gfCNCPoint5[3628] = {X 478.2330, Y 32.3647, Z -6.3333, A 0.000, B 0.000, C 0.000 }
gfCNCPoint5[3629] = {X 476.9689, Y 31.4976, Z -6.3333, A 0.000, B 0.000, C 0.000 }
gfCNCPoint5[3630] = {X 475.8319, Y 30.4695, Z -6.3333, A 0.000, B 0.000, C 0.000 }
gfCNCPoint5[3631] = {X 474.8423, Y 29.2987, Z -6.3333, A 0.000, B 0.000, C 0.000 }
gfCNCPoint5[3632] = {X 474.0180, Y 28.0063, Z -6.3333, A 0.000, B 0.000, C 0.000 }
gfCNCPoint5[3633] = {X 473.3736, Y 26.6154, Z -6.3333, A 0.000, B 0.000, C 0.000 }
gfCNCPoint5[3634] = {X 472.9207, Y 25.1509, Z -6.3333, A 0.000, B 0.000, C 0.000 }
gfCNCPoint5[3635] = {X 472.6068, Y 23.4678, Z -6.3333, A 0.000, B 0.000, C 0.000 }
gfCNCPoint5[3636] = {X 472.4665, Y 21.7615, Z -6.3333, A 0.000, B 0.000, C 0.000 }
gfCNCPoint5[3637] = {X 472.5012, Y 20.0497, Z -6.3333, A 0.000, B 0.000, C 0.000 }
gfCNCPoint5[3638] = {X 472.7106, Y 18.3505, Z -6.3333, A 0.000, B 0.000, C 0.000 }
gfCNCPoint5[3639] = {X 473.0925, Y 16.6815, Z -6.3333, A 0.000, B 0.000, C 0.000 }
gfCNCPoint5[3640] = {X 473.6354, Y 15.1666, Z -6.3333, A 0.000, B 0.000, C 0.000 }
gfCNCPoint5[3641] = {X 474.3788, Y 13.7394, Z -6.3333, A 0.000, B 0.000, C 0.000 }
gfCNCPoint5[3642] = {X 475.3090, Y 12.4262, Z -6.3333, A 0.000, B 0.000, C 0.000 }
gfCNCPoint5[3643] = {X 476.4087, Y 11.2513, Z -6.3333, A 0.000, B 0.000, C 0.000 }
gfCNCPoint5[3644] = {X 477.6577, Y 10.2366, Z -6.3333, A 0.000, B 0.000, C 0.000 }
gfCNCPoint5[3645] = {X 479.0328, Y 9.4006, Z -6.3333, A 0.000, B 0.000, C 0.000 }
gfCNCPoint5[3646] = {X 480.5086, Y 8.7590, Z -6.3333, A 0.000, B 0.000, C 0.000 }
gfCNCPoint5[3647] = {X 482.0578, Y 8.3236, Z -6.3333, A 0.000, B 0.000, C 0.000 }
gfCNCPoint5[3648] = {X 484.1552, Y 7.9970, Z -6.3333, A 0.000, B 0.000, C 0.000 }
gfCNCPoint5[3649] = {X 486.2746, Y 7.8821, Z -6.3333, A 0.000, B 0.000, C 0.000 }
gfCNCPoint5[3650] = {X 486.9679, Y 7.8699, Z -6.3333, A 0.000, B 0.000, C 0.000 }
gfCNCPoint5[3651] = {X 492.3835, Y 7.8699, Z -6.3333, A 0.000, B 0.000, C 0.000 }
gfCNCPoint5[3652] = {X 492.3835, Y 3.8699, Z -6.3333, A 0.000, B 0.000, C 0.000 }
gfCNCPoint5[3653] = {X 492.3835, Y 7.9499, Z -6.3333, A 0.000, B 0.000, C 0.000 }
gfCNCPoint5[3654] = {X 502.2063, Y 7.9499, Z -6.3333, A 0.000, B 0.000, C 0.000 }
gfCNCPoint5[3655] = {X 502.7389, Y 7.9541, Z -6.3333, A 0.000, B 0.000, C 0.000 }
gfCNCPoint5[3656] = {X 503.6731, Y 8.0662, Z -6.3333, A 0.000, B 0.000, C 0.000 }
gfCNCPoint5[3657] = {X 504.5592, Y 8.3824, Z -6.3333, A 0.000, B 0.000, C 0.000 }
gfCNCPoint5[3658] = {X 505.3534, Y 8.8870, Z -6.3333, A 0.000, B 0.000, C 0.000 }
gfCNCPoint5[3659] = {X 506.0160, Y 9.5548, Z -6.3333, A 0.000, B 0.000, C 0.000 }
gfCNCPoint5[3660] = {X 506.5144, Y 10.3529, Z -6.3333, A 0.000, B 0.000, C 0.000 }
gfCNCPoint5[3661] = {X 506.8237, Y 11.2415, Z -6.3333, A 0.000, B 0.000, C 0.000 }
gfCNCPoint5[3662] = {X 506.9285, Y 12.1765, Z -6.3333, A 0.000, B 0.000, C 0.000 }
gfCNCPoint5[3663] = {X 506.9285, Y 12.9782, Z -6.3333, A 0.000, B 0.000, C 0.000 }
gfCNCPoint5[3664] = {X 506.8271, Y 13.8997, Z -6.3333, A 0.000, B 0.000, C 0.000 }
gfCNCPoint5[3665] = {X 506.5279, Y 14.7771, Z -6.3333, A 0.000, B 0.000, C 0.000 }
gfCNCPoint5[3666] = {X 506.0451, Y 15.5686, Z -6.3333, A 0.000, B 0.000, C 0.000 }
gfCNCPoint5[3667] = {X 505.4018, Y 16.2362, Z -6.3333, A 0.000, B 0.000, C 0.000 }
gfCNCPoint5[3668] = {X 505.4017, Y 40.9510, Z -6.3333, A 0.000, B 0.000, C 0.000 }
gfCNCPoint5[3669] = {X 505.4300, Y 40.9743, Z -6.3333, A 0.000, B 0.000, C 0.000 }
gfCNCPoint5[3670] = {X 506.0563, Y 41.6329, Z -6.3333, A 0.000, B 0.000, C 0.000 }
gfCNCPoint5[3671] = {X 506.5279, Y 42.4098, Z -6.3333, A 0.000, B 0.000, C 0.000 }
gfCNCPoint5[3672] = {X 506.8231, Y 43.2693, Z -6.3333, A 0.000, B 0.000, C 0.000 }
gfCNCPoint5[3673] = {X 506.9283, Y 44.1720, Z -6.3333, A 0.000, B 0.000, C 0.000 }
gfCNCPoint5[3674] = {X 506.9285, Y 45.0000, Z -6.3333, A 0.000, B 0.000, C 0.000 }
gfCNCPoint5[3675] = {X 506.8222, Y 45.9435, Z -6.3333, A 0.000, B 0.000, C 0.000 }
gfCNCPoint5[3676] = {X 506.5086, Y 46.8397, Z -6.3333, A 0.000, B 0.000, C 0.000 }
gfCNCPoint5[3677] = {X 506.0035, Y 47.6436, Z -6.3333, A 0.000, B 0.000, C 0.000 }
gfCNCPoint5[3678] = {X 505.3321, Y 48.3150, Z -6.3333, A 0.000, B 0.000, C 0.000 }
gfCNCPoint5[3679] = {X 504.5282, Y 48.8201, Z -6.3333, A 0.000, B 0.000, C 0.000 }
gfCNCPoint5[3680] = {X 503.6320, Y 49.1337, Z -6.3333, A 0.000, B 0.000, C 0.000 }
gfCNCPoint5[3681] = {X 502.6885, Y 49.2400, Z -6.3333, A 0.000, B 0.000, C 0.000 }
gfCNCPoint5[3682] = {X 496.2450, Y 49.2400, Z -6.3333, A 0.000, B 0.000, C 0.000 }
gfCNCPoint5[3683] = {X 495.3062, Y 49.1348, Z -6.3333, A 0.000, B 0.000, C 0.000 }
gfCNCPoint5[3684] = {X 494.4140, Y 48.8242, Z -6.3333, A 0.000, B 0.000, C 0.000 }
gfCNCPoint5[3685] = {X 493.6127, Y 48.3239, Z -6.3333, A 0.000, B 0.000, C 0.000 }
gfCNCPoint5[3686] = {X 492.9420, Y 47.6585, Z -6.3333, A 0.000, B 0.000, C 0.000 }
gfCNCPoint5[3687] = {X 492.4354, Y 46.8612, Z -6.3333, A 0.000, B 0.000, C 0.000 }
gfCNCPoint5[3688] = {X 492.1178, Y 45.9714, Z -6.3333, A 0.000, B 0.000, C 0.000 }
gfCNCPoint5[3689] = {X 492.0052, Y 45.0335, Z -6.3333, A 0.000, B 0.000, C 0.000 }
gfCNCPoint5[3690] = {X 492.0054, Y 44.1505, Z -6.3333, A 0.000, B 0.000, C 0.000 }
gfCNCPoint5[3691] = {X 492.1159, Y 43.2454, Z -6.3333, A 0.000, B 0.000, C 0.000 }
gfCNCPoint5[3692] = {X 492.4173, Y 42.3850, Z -6.3333, A 0.000, B 0.000, C 0.000 }
gfCNCPoint5[3693] = {X 492.8957, Y 41.6088, Z -6.3333, A 0.000, B 0.000, C 0.000 }
gfCNCPoint5[3694] = {X 493.5290, Y 40.9529, Z -6.3333, A 0.000, B 0.000, C 0.000 }
gfCNCPoint5[3695] = {X 493.5290, Y 34.3938, Z -6.3333, A 0.000, B 0.000, C 0.000 }
gfCNCPoint5[3696] = {X 490.6762, Y 34.3938, Z -6.3333, A 0.000, B 0.000, C 0.000 }
gfCNCPoint5[3697] = {X 486.3532, Y 42.8123, Z -6.3333, A 0.000, B 0.000, C 0.000 }
gfCNCPoint5[3698] = {X 486.3698, Y 42.8571, Z -6.3333, A 0.000, B 0.000, C 0.000 }
gfCNCPoint5[3699] = {X 486.5322, Y 43.5051, Z -6.3333, A 0.000, B 0.000, C 0.000 }
gfCNCPoint5[3700] = {X 486.5908, Y 44.1706, Z -6.3333, A 0.000, B 0.000, C 0.000 }
gfCNCPoint5[3701] = {X 486.5910, Y 45.0000, Z -6.3333, A 0.000, B 0.000, C 0.000 }
gfCNCPoint5[3702] = {X 486.4847, Y 45.9435, Z -6.3333, A 0.000, B 0.000, C 0.000 }
gfCNCPoint5[3703] = {X 486.1711, Y 46.8397, Z -6.3333, A 0.000, B 0.000, C 0.000 }
gfCNCPoint5[3704] = {X 485.6660, Y 47.6436, Z -6.3333, A 0.000, B 0.000, C 0.000 }
gfCNCPoint5[3705] = {X 484.9946, Y 48.3150, Z -6.3333, A 0.000, B 0.000, C 0.000 }
gfCNCPoint5[3706] = {X 484.1907, Y 48.8201, Z -6.3333, A 0.000, B 0.000, C 0.000 }
gfCNCPoint5[3707] = {X 483.2945, Y 49.1337, Z -6.3333, A 0.000, B 0.000, C 0.000 }
gfCNCPoint5[3708] = {X 482.3510, Y 49.2400, Z -6.3333, A 0.000, B 0.000, C 0.000 }
gfCNCPoint5[3709] = {X 475.7650, Y 49.2400, Z -6.3333, A 0.000, B 0.000, C 0.000 }
gfCNCPoint5[3710] = {X 474.8215, Y 49.1337, Z -6.3333, A 0.000, B 0.000, C 0.000 }
gfCNCPoint5[3711] = {X 473.9253, Y 48.8201, Z -6.3333, A 0.000, B 0.000, C 0.000 }
gfCNCPoint5[3712] = {X 473.1214, Y 48.3150, Z -6.3333, A 0.000, B 0.000, C 0.000 }
gfCNCPoint5[3713] = {X 472.4500, Y 47.6436, Z -6.3333, A 0.000, B 0.000, C 0.000 }
gfCNCPoint5[3714] = {X 471.9449, Y 46.8397, Z -6.3333, A 0.000, B 0.000, C 0.000 }
gfCNCPoint5[3715] = {X 471.6313, Y 45.9436, Z -6.3333, A 0.000, B 0.000, C 0.000 }
gfCNCPoint5[3716] = {X 471.5250, Y 45.0001, Z -6.3333, A 0.000, B 0.000, C 0.000 }
gfCNCPoint5[3717] = {X 471.5254, Y 44.1505, Z -6.3333, A 0.000, B 0.000, C 0.000 }
gfCNCPoint5[3718] = {X 471.6223, Y 43.3054, Z -6.3333, A 0.000, B 0.000, C 0.000 }
gfCNCPoint5[3719] = {X 471.8860, Y 42.4967, Z -6.3333, A 0.000, B 0.000, C 0.000 }
gfCNCPoint5[3720] = {X 472.3057, Y 41.7570, Z -6.3333, A 0.000, B 0.000, C 0.000 }
gfCNCPoint5[3721] = {X 472.8647, Y 41.1159, Z -6.3333, A 0.000, B 0.000, C 0.000 }
gfCNCPoint5[3722] = {X 473.5404, Y 40.5992, Z -6.3333, A 0.000, B 0.000, C 0.000 }
gfCNCPoint5[3723] = {X 474.3057, Y 40.2278, Z -6.3333, A 0.000, B 0.000, C 0.000 }
gfCNCPoint5[3724] = {X 478.3385, Y 32.3339, Z -6.3333, A 0.000, B 0.000, C 0.000 }
gfCNCPoint5[3725] = {X 477.0677, Y 31.4735, Z -6.3333, A 0.000, B 0.000, C 0.000 }
gfCNCPoint5[3726] = {X 475.9242, Y 30.4498, Z -6.3333, A 0.000, B 0.000, C 0.000 }
gfCNCPoint5[3727] = {X 474.9290, Y 29.2814, Z -6.3333, A 0.000, B 0.000, C 0.000 }
gfCNCPoint5[3728] = {X 474.1002, Y 27.9898, Z -6.3333, A 0.000, B 0.000, C 0.000 }
gfCNCPoint5[3729] = {X 473.4527, Y 26.5983, Z -6.3333, A 0.000, B 0.000, C 0.000 }
gfCNCPoint5[3730] = {X 472.9985, Y 25.1323, Z -6.3333, A 0.000, B 0.000, C 0.000 }
gfCNCPoint5[3731] = {X 472.6861, Y 23.4572, Z -6.3333, A 0.000, B 0.000, C 0.000 }
gfCNCPoint5[3732] = {X 472.5465, Y 21.7590, Z -6.3333, A 0.000, B 0.000, C 0.000 }
gfCNCPoint5[3733] = {X 472.5810, Y 20.0555, Z -6.3333, A 0.000, B 0.000, C 0.000 }
gfCNCPoint5[3734] = {X 472.7894, Y 18.3643, Z -6.3333, A 0.000, B 0.000, C 0.000 }
gfCNCPoint5[3735] = {X 473.1695, Y 16.7033, Z -6.3333, A 0.000, B 0.000, C 0.000 }
gfCNCPoint5[3736] = {X 473.7087, Y 15.1986, Z -6.3333, A 0.000, B 0.000, C 0.000 }
gfCNCPoint5[3737] = {X 474.4471, Y 13.7811, Z -6.3333, A 0.000, B 0.000, C 0.000 }
gfCNCPoint5[3738] = {X 475.3710, Y 12.4767, Z -6.3333, A 0.000, B 0.000, C 0.000 }
gfCNCPoint5[3739] = {X 476.4633, Y 11.3098, Z -6.3333, A 0.000, B 0.000, C 0.000 }
gfCNCPoint5[3740] = {X 477.7038, Y 10.3019, Z -6.3333, A 0.000, B 0.000, C 0.000 }
gfCNCPoint5[3741] = {X 479.0696, Y 9.4717, Z -6.3333, A 0.000, B 0.000, C 0.000 }
gfCNCPoint5[3742] = {X 480.5355, Y 8.8344, Z -6.3333, A 0.000, B 0.000, C 0.000 }
gfCNCPoint5[3743] = {X 482.0742, Y 8.4019, Z -6.3333, A 0.000, B 0.000, C 0.000 }
gfCNCPoint5[3744] = {X 484.1638, Y 8.0765, Z -6.3333, A 0.000, B 0.000, C 0.000 }
gfCNCPoint5[3745] = {X 486.2755, Y 7.9621, Z -6.3333, A 0.000, B 0.000, C 0.000 }
gfCNCPoint5[3746] = {X 486.9686, Y 7.9499, Z -6.3333, A 0.000, B 0.000, C 0.000 }
gfCNCPoint5[3747] = {X 492.3835, Y 7.9499, Z -6.3333, A 0.000, B 0.000, C 0.000 }
gfCNCPoint5[3748] = {X 492.3835, Y 3.9499, Z -6.3333, A 0.000, B 0.000, C 0.000 }
gfCNCPoint5[3749] = {X 492.3835, Y 8.0299, Z -6.3333, A 0.000, B 0.000, C 0.000 }
gfCNCPoint5[3750] = {X 502.2059, Y 8.0299, Z -6.3333, A 0.000, B 0.000, C 0.000 }
gfCNCPoint5[3751] = {X 502.7383, Y 8.0341, Z -6.3333, A 0.000, B 0.000, C 0.000 }
gfCNCPoint5[3752] = {X 503.6547, Y 8.1441, Z -6.3333, A 0.000, B 0.000, C 0.000 }
gfCNCPoint5[3753] = {X 504.5241, Y 8.4543, Z -6.3333, A 0.000, B 0.000, C 0.000 }
gfCNCPoint5[3754] = {X 505.3032, Y 8.9493, Z -6.3333, A 0.000, B 0.000, C 0.000 }
gfCNCPoint5[3755] = {X 505.9533, Y 9.6045, Z -6.3333, A 0.000, B 0.000, C 0.000 }
gfCNCPoint5[3756] = {X 506.4422, Y 10.3875, Z -6.3333, A 0.000, B 0.000, C 0.000 }
gfCNCPoint5[3757] = {X 506.7457, Y 11.2592, Z -6.3333, A 0.000, B 0.000, C 0.000 }
gfCNCPoint5[3758] = {X 506.8485, Y 12.1765, Z -6.3333, A 0.000, B 0.000, C 0.000 }
gfCNCPoint5[3759] = {X 506.8485, Y 12.9782, Z -6.3333, A 0.000, B 0.000, C 0.000 }
gfCNCPoint5[3760] = {X 506.7470, Y 13.8914, Z -6.3333, A 0.000, B 0.000, C 0.000 }
gfCNCPoint5[3761] = {X 506.4475, Y 14.7601, Z -6.3333, A 0.000, B 0.000, C 0.000 }
gfCNCPoint5[3762] = {X 505.9645, Y 15.5418, Z -6.3333, A 0.000, B 0.000, C 0.000 }
gfCNCPoint5[3763] = {X 505.3218, Y 16.1985, Z -6.3333, A 0.000, B 0.000, C 0.000 }
gfCNCPoint5[3764] = {X 505.3217, Y 40.9891, Z -6.3333, A 0.000, B 0.000, C 0.000 }
gfCNCPoint5[3765] = {X 505.3681, Y 41.0268, Z -6.3333, A 0.000, B 0.000, C 0.000 }
gfCNCPoint5[3766] = {X 505.9867, Y 41.6736, Z -6.3333, A 0.000, B 0.000, C 0.000 }
gfCNCPoint5[3767] = {X 506.4526, Y 42.4377, Z -6.3333, A 0.000, B 0.000, C 0.000 }
gfCNCPoint5[3768] = {X 506.7443, Y 43.2838, Z -6.3333, A 0.000, B 0.000, C 0.000 }
gfCNCPoint5[3769] = {X 506.8483, Y 44.1727, Z -6.3333, A 0.000, B 0.000, C 0.000 }
gfCNCPoint5[3770] = {X 506.8485, Y 45.0000, Z -6.3333, A 0.000, B 0.000, C 0.000 }
gfCNCPoint5[3771] = {X 506.7442, Y 45.9257, Z -6.3333, A 0.000, B 0.000, C 0.000 }
gfCNCPoint5[3772] = {X 506.4365, Y 46.8050, Z -6.3333, A 0.000, B 0.000, C 0.000 }
gfCNCPoint5[3773] = {X 505.9409, Y 47.5937, Z -6.3333, A 0.000, B 0.000, C 0.000 }
gfCNCPoint5[3774] = {X 505.2822, Y 48.2524, Z -6.3333, A 0.000, B 0.000, C 0.000 }
gfCNCPoint5[3775] = {X 504.4934, Y 48.7480, Z -6.3333, A 0.000, B 0.000, C 0.000 }
gfCNCPoint5[3776] = {X 503.6142, Y 49.0557, Z -6.3333, A 0.000, B 0.000, C 0.000 }
gfCNCPoint5[3777] = {X 502.6885, Y 49.1600, Z -6.3333, A 0.000, B 0.000, C 0.000 }
gfCNCPoint5[3778] = {X 496.2450, Y 49.1600, Z -6.3333, A 0.000, B 0.000, C 0.000 }
gfCNCPoint5[3779] = {X 495.3239, Y 49.0567, Z -6.3333, A 0.000, B 0.000, C 0.000 }
gfCNCPoint5[3780] = {X 494.4485, Y 48.7521, Z -6.3333, A 0.000, B 0.000, C 0.000 }
gfCNCPoint5[3781] = {X 493.6623, Y 48.2612, Z -6.3333, A 0.000, B 0.000, C 0.000 }
gfCNCPoint5[3782] = {X 493.0043, Y 47.6084, Z -6.3333, A 0.000, B 0.000, C 0.000 }
gfCNCPoint5[3783] = {X 492.5072, Y 46.8261, Z -6.3333, A 0.000, B 0.000, C 0.000 }
gfCNCPoint5[3784] = {X 492.1957, Y 45.9531, Z -6.3333, A 0.000, B 0.000, C 0.000 }
gfCNCPoint5[3785] = {X 492.0852, Y 45.0328, Z -6.3333, A 0.000, B 0.000, C 0.000 }
gfCNCPoint5[3786] = {X 492.0854, Y 44.1516, Z -6.3333, A 0.000, B 0.000, C 0.000 }
gfCNCPoint5[3787] = {X 492.1960, Y 43.2545, Z -6.3333, A 0.000, B 0.000, C 0.000 }
gfCNCPoint5[3788] = {X 492.4976, Y 42.4026, Z -6.3333, A 0.000, B 0.000, C 0.000 }
gfCNCPoint5[3789] = {X 492.9762, Y 41.6358, Z -6.3333, A 0.000, B 0.000, C 0.000 }
gfCNCPoint5[3790] = {X 493.6090, Y 40.9906, Z -6.3333, A 0.000, B 0.000, C 0.000 }
gfCNCPoint5[3791] = {X 493.6090, Y 34.3138, Z -6.3333, A 0.000, B 0.000, C 0.000 }
gfCNCPoint5[3792] = {X 490.6274, Y 34.3138, Z -6.3333, A 0.000, B 0.000, C 0.000 }
gfCNCPoint5[3793] = {X 486.2660, Y 42.8071, Z -6.3333, A 0.000, B 0.000, C 0.000 }
gfCNCPoint5[3794] = {X 486.2944, Y 42.8838, Z -6.3333, A 0.000, B 0.000, C 0.000 }
gfCNCPoint5[3795] = {X 486.4534, Y 43.5190, Z -6.3333, A 0.000, B 0.000, C 0.000 }
gfCNCPoint5[3796] = {X 486.5108, Y 44.1713, Z -6.3333, A 0.000, B 0.000, C 0.000 }
gfCNCPoint5[3797] = {X 486.5110, Y 45.0000, Z -6.3333, A 0.000, B 0.000, C 0.000 }
gfCNCPoint5[3798] = {X 486.4067, Y 45.9257, Z -6.3333, A 0.000, B 0.000, C 0.000 }
gfCNCPoint5[3799] = {X 486.0990, Y 46.8050, Z -6.3333, A 0.000, B 0.000, C 0.000 }
gfCNCPoint5[3800] = {X 485.6034, Y 47.5937, Z -6.3333, A 0.000, B 0.000, C 0.000 }
gfCNCPoint5[3801] = {X 484.9447, Y 48.2524, Z -6.3333, A 0.000, B 0.000, C 0.000 }
gfCNCPoint5[3802] = {X 484.1560, Y 48.7480, Z -6.3333, A 0.000, B 0.000, C 0.000 }
gfCNCPoint5[3803] = {X 483.2767, Y 49.0557, Z -6.3333, A 0.000, B 0.000, C 0.000 }
gfCNCPoint5[3804] = {X 482.3510, Y 49.1600, Z -6.3333, A 0.000, B 0.000, C 0.000 }
gfCNCPoint5[3805] = {X 475.7650, Y 49.1600, Z -6.3333, A 0.000, B 0.000, C 0.000 }
gfCNCPoint5[3806] = {X 474.8393, Y 49.0557, Z -6.3333, A 0.000, B 0.000, C 0.000 }
gfCNCPoint5[3807] = {X 473.9600, Y 48.7480, Z -6.3333, A 0.000, B 0.000, C 0.000 }
gfCNCPoint5[3808] = {X 473.1713, Y 48.2524, Z -6.3333, A 0.000, B 0.000, C 0.000 }
gfCNCPoint5[3809] = {X 472.5126, Y 47.5937, Z -6.3333, A 0.000, B 0.000, C 0.000 }
gfCNCPoint5[3810] = {X 472.0169, Y 46.8050, Z -6.3333, A 0.000, B 0.000, C 0.000 }
gfCNCPoint5[3811] = {X 471.7093, Y 45.9257, Z -6.3333, A 0.000, B 0.000, C 0.000 }
gfCNCPoint5[3812] = {X 471.6050, Y 45.0000, Z -6.3333, A 0.000, B 0.000, C 0.000 }
gfCNCPoint5[3813] = {X 471.6054, Y 44.1516, Z -6.3333, A 0.000, B 0.000, C 0.000 }
gfCNCPoint5[3814] = {X 471.7016, Y 43.3174, Z -6.3333, A 0.000, B 0.000, C 0.000 }
gfCNCPoint5[3815] = {X 471.9634, Y 42.5195, Z -6.3333, A 0.000, B 0.000, C 0.000 }
gfCNCPoint5[3816] = {X 472.3801, Y 41.7905, Z -6.3333, A 0.000, B 0.000, C 0.000 }
gfCNCPoint5[3817] = {X 472.9347, Y 41.1600, Z -6.3333, A 0.000, B 0.000, C 0.000 }
gfCNCPoint5[3818] = {X 473.6046, Y 40.6537, Z -6.3333, A 0.000, B 0.000, C 0.000 }
gfCNCPoint5[3819] = {X 474.3626, Y 40.2923, Z -6.3333, A 0.000, B 0.000, C 0.000 }
gfCNCPoint5[3820] = {X 478.4443, Y 32.3027, Z -6.3333, A 0.000, B 0.000, C 0.000 }
gfCNCPoint5[3821] = {X 477.1667, Y 31.4491, Z -6.3333, A 0.000, B 0.000, C 0.000 }
gfCNCPoint5[3822] = {X 476.0168, Y 30.4299, Z -6.3333, A 0.000, B 0.000, C 0.000 }
gfCNCPoint5[3823] = {X 475.0159, Y 29.2641, Z -6.3333, A 0.000, B 0.000, C 0.000 }
gfCNCPoint5[3824] = {X 474.1824, Y 27.9733, Z -6.3333, A 0.000, B 0.000, C 0.000 }
gfCNCPoint5[3825] = {X 473.5319, Y 26.5812, Z -6.3333, A 0.000, B 0.000, C 0.000 }
gfCNCPoint5[3826] = {X 473.0764, Y 25.1137, Z -6.3333, A 0.000, B 0.000, C 0.000 }
gfCNCPoint5[3827] = {X 472.7654, Y 23.4467, Z -6.3333, A 0.000, B 0.000, C 0.000 }
gfCNCPoint5[3828] = {X 472.6264, Y 21.7567, Z -6.3333, A 0.000, B 0.000, C 0.000 }
gfCNCPoint5[3829] = {X 472.6608, Y 20.0612, Z -6.3333, A 0.000, B 0.000, C 0.000 }
gfCNCPoint5[3830] = {X 472.8682, Y 18.3782, Z -6.3333, A 0.000, B 0.000, C 0.000 }
gfCNCPoint5[3831] = {X 473.2464, Y 16.7251, Z -6.3333, A 0.000, B 0.000, C 0.000 }
gfCNCPoint5[3832] = {X 473.7820, Y 15.2307, Z -6.3333, A 0.000, B 0.000, C 0.000 }
gfCNCPoint5[3833] = {X 474.5153, Y 13.8227, Z -6.3333, A 0.000, B 0.000, C 0.000 }
gfCNCPoint5[3834] = {X 475.4330, Y 12.5273, Z -6.3333, A 0.000, B 0.000, C 0.000 }
gfCNCPoint5[3835] = {X 476.5178, Y 11.3684, Z -6.3333, A 0.000, B 0.000, C 0.000 }
gfCNCPoint5[3836] = {X 477.7499, Y 10.3673, Z -6.3333, A 0.000, B 0.000, C 0.000 }
gfCNCPoint5[3837] = {X 479.1064, Y 9.5427, Z -6.3333, A 0.000, B 0.000, C 0.000 }
gfCNCPoint5[3838] = {X 480.5623, Y 8.9097, Z -6.3333, A 0.000, B 0.000, C 0.000 }
gfCNCPoint5[3839] = {X 482.0906, Y 8.4802, Z -6.3333, A 0.000, B 0.000, C 0.000 }
gfCNCPoint5[3840] = {X 484.1725, Y 8.1560, Z -6.3333, A 0.000, B 0.000, C 0.000 }
gfCNCPoint5[3841] = {X 486.2764, Y 8.0421, Z -6.3333, A 0.000, B 0.000, C 0.000 }
gfCNCPoint5[3842] = {X 486.9693, Y 8.0299, Z -6.3333, A 0.000, B 0.000, C 0.000 }
gfCNCPoint5[3843] = {X 492.3835, Y 8.0299, Z -6.3333, A 0.000, B 0.000, C 0.000 }
gfCNCPoint5[3844] = {X 492.3835, Y 4.0299, Z -6.3333, A 0.000, B 0.000, C 0.000 }
gfCNCPoint5[3845] = {X 492.3835, Y 8.1099, Z -6.3333, A 0.000, B 0.000, C 0.000 }
gfCNCPoint5[3846] = {X 502.2056, Y 8.1099, Z -6.3333, A 0.000, B 0.000, C 0.000 }
gfCNCPoint5[3847] = {X 502.7376, Y 8.1141, Z -6.3333, A 0.000, B 0.000, C 0.000 }
gfCNCPoint5[3848] = {X 503.6364, Y 8.2219, Z -6.3333, A 0.000, B 0.000, C 0.000 }
gfCNCPoint5[3849] = {X 504.4890, Y 8.5261, Z -6.3333, A 0.000, B 0.000, C 0.000 }
gfCNCPoint5[3850] = {X 505.2530, Y 9.0116, Z -6.3333, A 0.000, B 0.000, C 0.000 }
gfCNCPoint5[3851] = {X 505.8906, Y 9.6542, Z -6.3333, A 0.000, B 0.000, C 0.000 }
gfCNCPoint5[3852] = {X 506.3701, Y 10.4220, Z -6.3333, A 0.000, B 0.000, C 0.000 }
gfCNCPoint5[3853] = {X 506.6676, Y 11.2769, Z -6.3333, A 0.000, B 0.000, C 0.000 }
gfCNCPoint5[3854] = {X 506.7685, Y 12.1765, Z -6.3333, A 0.000, B 0.000, C 0.000 }
gfCNCPoint5[3855] = {X 506.7685, Y 12.9782, Z -6.3333, A 0.000, B 0.000, C 0.000 }
gfCNCPoint5[3856] = {X 506.6668, Y 13.8831, Z -6.3333, A 0.000, B 0.000, C 0.000 }
gfCNCPoint5[3857] = {X 506.3670, Y 14.7429, Z -6.3333, A 0.000, B 0.000, C 0.000 }
gfCNCPoint5[3858] = {X 505.8840, Y 15.5148, Z -6.3333, A 0.000, B 0.000, C 0.000 }
gfCNCPoint5[3859] = {X 505.2418, Y 16.1603, Z -6.3333, A 0.000, B 0.000, C 0.000 }
gfCNCPoint5[3860] = {X 505.2417, Y 41.0271, Z -6.3333, A 0.000, B 0.000, C 0.000 }
gfCNCPoint5[3861] = {X 505.3177, Y 41.0889, Z -6.3333, A 0.000, B 0.000, C 0.000 }
gfCNCPoint5[3862] = {X 505.9239, Y 41.7232, Z -6.3333, A 0.000, B 0.000, C 0.000 }
gfCNCPoint5[3863] = {X 506.3805, Y 42.4724, Z -6.3333, A 0.000, B 0.000, C 0.000 }
gfCNCPoint5[3864] = {X 506.6664, Y 43.3019, Z -6.3333, A 0.000, B 0.000, C 0.000 }
gfCNCPoint5[3865] = {X 506.7683, Y 44.1734, Z -6.3333, A 0.000, B 0.000, C 0.000 }
gfCNCPoint5[3866] = {X 506.7685, Y 45.0000, Z -6.3333, A 0.000, B 0.000, C 0.000 }
gfCNCPoint5[3867] = {X 506.6662, Y 45.9079, Z -6.3333, A 0.000, B 0.000, C 0.000 }
gfCNCPoint5[3868] = {X 506.3644, Y 46.7702, Z -6.3333, A 0.000, B 0.000, C 0.000 }
gfCNCPoint5[3869] = {X 505.8784, Y 47.5438, Z -6.3333, A 0.000, B 0.000, C 0.000 }
gfCNCPoint5[3870] = {X 505.2323, Y 48.1899, Z -6.3333, A 0.000, B 0.000, C 0.000 }
gfCNCPoint5[3871] = {X 504.4587, Y 48.6760, Z -6.3333, A 0.000, B 0.000, C 0.000 }
gfCNCPoint5[3872] = {X 503.5964, Y 48.9777, Z -6.3333, A 0.000, B 0.000, C 0.000 }
gfCNCPoint5[3873] = {X 502.6885, Y 49.0800, Z -6.3333, A 0.000, B 0.000, C 0.000 }
gfCNCPoint5[3874] = {X 496.2450, Y 49.0800, Z -6.3333, A 0.000, B 0.000, C 0.000 }
gfCNCPoint5[3875] = {X 495.3416, Y 48.9787, Z -6.3333, A 0.000, B 0.000, C 0.000 }
gfCNCPoint5[3876] = {X 494.4831, Y 48.6799, Z -6.3333, A 0.000, B 0.000, C 0.000 }
gfCNCPoint5[3877] = {X 493.7120, Y 48.1985, Z -6.3333, A 0.000, B 0.000, C 0.000 }
gfCNCPoint5[3878] = {X 493.0667, Y 47.5582, Z -6.3333, A 0.000, B 0.000, C 0.000 }
gfCNCPoint5[3879] = {X 492.5791, Y 46.7909, Z -6.3333, A 0.000, B 0.000, C 0.000 }
gfCNCPoint5[3880] = {X 492.2736, Y 45.9348, Z -6.3333, A 0.000, B 0.000, C 0.000 }
gfCNCPoint5[3881] = {X 492.1652, Y 45.0322, Z -6.3333, A 0.000, B 0.000, C 0.000 }
gfCNCPoint5[3882] = {X 492.1654, Y 44.1527, Z -6.3333, A 0.000, B 0.000, C 0.000 }
gfCNCPoint5[3883] = {X 492.2760, Y 43.2637, Z -6.3333, A 0.000, B 0.000, C 0.000 }
gfCNCPoint5[3884] = {X 492.5779, Y 42.4203, Z -6.3333, A 0.000, B 0.000, C 0.000 }
gfCNCPoint5[3885] = {X 493.0566, Y 41.6631, Z -6.3333, A 0.000, B 0.000, C 0.000 }
gfCNCPoint5[3886] = {X 493.6890, Y 41.0287, Z -6.3333, A 0.000, B 0.000, C 0.000 }
gfCNCPoint5[3887] = {X 493.6890, Y 34.2338, Z -6.3333, A 0.000, B 0.000, C 0.000 }
gfCNCPoint5[3888] = {X 490.5785, Y 34.2338, Z -6.3333, A 0.000, B 0.000, C 0.000 }
gfCNCPoint5[3889] = {X 486.1787, Y 42.8019, Z -6.3333, A 0.000, B 0.000, C 0.000 }
gfCNCPoint5[3890] = {X 486.2189, Y 42.9104, Z -6.3333, A 0.000, B 0.000, C 0.000 }
gfCNCPoint5[3891] = {X 486.3746, Y 43.5329, Z -6.3333, A 0.000, B 0.000, C 0.000 }
gfCNCPoint5[3892] = {X 486.4309, Y 44.1720, Z -6.3333, A 0.000, B 0.000, C 0.000 }
gfCNCPoint5[3893] = {X 486.4310, Y 45.0000, Z -6.3333, A 0.000, B 0.000, C 0.000 }
gfCNCPoint5[3894] = {X 486.3287, Y 45.9079, Z -6.3333, A 0.000, B 0.000, C 0.000 }
gfCNCPoint5[3895] = {X 486.0270, Y 46.7702, Z -6.3333, A 0.000, B 0.000, C 0.000 }
gfCNCPoint5[3896] = {X 485.5409, Y 47.5438, Z -6.3333, A 0.000, B 0.000, C 0.000 }
gfCNCPoint5[3897] = {X 484.8949, Y 48.1899, Z -6.3333, A 0.000, B 0.000, C 0.000 }
gfCNCPoint5[3898] = {X 484.1213, Y 48.6760, Z -6.3333, A 0.000, B 0.000, C 0.000 }
gfCNCPoint5[3899] = {X 483.2589, Y 48.9777, Z -6.3333, A 0.000, B 0.000, C 0.000 }
gfCNCPoint5[3900] = {X 482.3510, Y 49.0800, Z -6.3333, A 0.000, B 0.000, C 0.000 }
gfCNCPoint5[3901] = {X 475.7650, Y 49.0800, Z -6.3333, A 0.000, B 0.000, C 0.000 }
gfCNCPoint5[3902] = {X 474.8571, Y 48.9777, Z -6.3333, A 0.000, B 0.000, C 0.000 }
gfCNCPoint5[3903] = {X 473.9947, Y 48.6760, Z -6.3333, A 0.000, B 0.000, C 0.000 }
gfCNCPoint5[3904] = {X 473.2211, Y 48.1899, Z -6.3333, A 0.000, B 0.000, C 0.000 }
gfCNCPoint5[3905] = {X 472.5751, Y 47.5438, Z -6.3333, A 0.000, B 0.000, C 0.000 }
gfCNCPoint5[3906] = {X 472.0890, Y 46.7702, Z -6.3333, A 0.000, B 0.000, C 0.000 }
gfCNCPoint5[3907] = {X 471.7873, Y 45.9079, Z -6.3333, A 0.000, B 0.000, C 0.000 }
gfCNCPoint5[3908] = {X 471.6850, Y 45.0000, Z -6.3333, A 0.000, B 0.000, C 0.000 }
gfCNCPoint5[3909] = {X 471.6853, Y 44.1527, Z -6.3333, A 0.000, B 0.000, C 0.000 }
gfCNCPoint5[3910] = {X 471.7809, Y 43.3294, Z -6.3333, A 0.000, B 0.000, C 0.000 }
gfCNCPoint5[3911] = {X 472.0408, Y 42.5424, Z -6.3333, A 0.000, B 0.000, C 0.000 }
gfCNCPoint5[3912] = {X 472.4544, Y 41.8242, Z -6.3333, A 0.000, B 0.000, C 0.000 }
gfCNCPoint5[3913] = {X 473.0046, Y 41.2044, Z -6.3333, A 0.000, B 0.000, C 0.000 }
gfCNCPoint5[3914] = {X 473.6687, Y 40.7085, Z -6.3333, A 0.000, B 0.000, C 0.000 }
gfCNCPoint5[3915] = {X 474.4193, Y 40.3571, Z -6.3333, A 0.000, B 0.000, C 0.000 }
gfCNCPoint5[3916] = {X 478.5503, Y 32.2710, Z -6.3333, A 0.000, B 0.000, C 0.000 }
gfCNCPoint5[3917] = {X 477.2659, Y 31.4244, Z -6.3333, A 0.000, B 0.000, C 0.000 }
gfCNCPoint5[3918] = {X 476.1095, Y 30.4099, Z -6.3333, A 0.000, B 0.000, C 0.000 }
gfCNCPoint5[3919] = {X 475.1028, Y 29.2467, Z -6.3333, A 0.000, B 0.000, C 0.000 }
gfCNCPoint5[3920] = {X 474.2647, Y 27.9567, Z -6.3333, A 0.000, B 0.000, C 0.000 }
gfCNCPoint5[3921] = {X 473.6111, Y 26.5641, Z -6.3333, A 0.000, B 0.000, C 0.000 }
gfCNCPoint5[3922] = {X 473.1542, Y 25.0952, Z -6.3333, A 0.000, B 0.000, C 0.000 }
gfCNCPoint5[3923] = {X 472.8448, Y 23.4362, Z -6.3333, A 0.000, B 0.000, C 0.000 }
gfCNCPoint5[3924] = {X 472.7064, Y 21.7543, Z -6.3333, A 0.000, B 0.000, C 0.000 }
gfCNCPoint5[3925] = {X 472.7406, Y 20.0670, Z -6.3333, A 0.000, B 0.000, C 0.000 }
gfCNCPoint5[3926] = {X 472.9470, Y 18.3920, Z -6.3333, A 0.000, B 0.000, C 0.000 }
gfCNCPoint5[3927] = {X 473.3234, Y 16.7469, Z -6.3333, A 0.000, B 0.000, C 0.000 }
gfCNCPoint5[3928] = {X 473.8553, Y 15.2627, Z -6.3333, A 0.000, B 0.000, C 0.000 }
gfCNCPoint5[3929] = {X 474.5836, Y 13.8644, Z -6.3333, A 0.000, B 0.000, C 0.000 }
gfCNCPoint5[3930] = {X 475.4949, Y 12.5779, Z -6.3333, A 0.000, B 0.000, C 0.000 }
gfCNCPoint5[3931] = {X 476.5724, Y 11.4269, Z -6.3333, A 0.000, B 0.000, C 0.000 }
gfCNCPoint5[3932] = {X 477.7960, Y 10.4327, Z -6.3333, A 0.000, B 0.000, C 0.000 }
gfCNCPoint5[3933] = {X 479.1432, Y 9.6137, Z -6.3333, A 0.000, B 0.000, C 0.000 }
gfCNCPoint5[3934] = {X 480.5891, Y 8.9851, Z -6.3333, A 0.000, B 0.000, C 0.000 }
gfCNCPoint5[3935] = {X 482.1069, Y 8.5585, Z -6.3333, A 0.000, B 0.000, C 0.000 }
gfCNCPoint5[3936] = {X 484.1812, Y 8.2356, Z -6.3333, A 0.000, B 0.000, C 0.000 }
gfCNCPoint5[3937] = {X 486.2773, Y 8.1221, Z -6.3333, A 0.000, B 0.000, C 0.000 }
gfCNCPoint5[3938] = {X 486.9700, Y 8.1099, Z -6.3333, A 0.000, B 0.000, C 0.000 }
gfCNCPoint5[3939] = {X 492.3835, Y 8.1099, Z -6.3333, A 0.000, B 0.000, C 0.000 }
gfCNCPoint5[3940] = {X 492.3835, Y 4.1099, Z -6.3333, A 0.000, B 0.000, C 0.000 }
gfCNCPoint5[3941] = {X 492.3835, Y 8.1899, Z -6.3333, A 0.000, B 0.000, C 0.000 }
gfCNCPoint5[3942] = {X 502.2053, Y 8.1899, Z -6.3333, A 0.000, B 0.000, C 0.000 }
gfCNCPoint5[3943] = {X 502.7370, Y 8.1941, Z -6.3333, A 0.000, B 0.000, C 0.000 }
gfCNCPoint5[3944] = {X 503.6181, Y 8.2998, Z -6.3333, A 0.000, B 0.000, C 0.000 }
gfCNCPoint5[3945] = {X 504.4539, Y 8.5980, Z -6.3333, A 0.000, B 0.000, C 0.000 }
gfCNCPoint5[3946] = {X 505.2029, Y 9.0739, Z -6.3333, A 0.000, B 0.000, C 0.000 }
gfCNCPoint5[3947] = {X 505.8279, Y 9.7039, Z -6.3333, A 0.000, B 0.000, C 0.000 }
gfCNCPoint5[3948] = {X 506.2979, Y 10.4566, Z -6.3333, A 0.000, B 0.000, C 0.000 }
gfCNCPoint5[3949] = {X 506.5896, Y 11.2946, Z -6.3333, A 0.000, B 0.000, C 0.000 }
gfCNCPoint5[3950] = {X 506.6885, Y 12.1765, Z -6.3333, A 0.000, B 0.000, C 0.000 }
gfCNCPoint5[3951] = {X 506.6883, Y 13.0192, Z -6.3333, A 0.000, B 0.000, C 0.000 }
gfCNCPoint5[3952] = {X 506.5797, Y 13.9046, Z -6.3333, A 0.000, B 0.000, C 0.000 }
gfCNCPoint5[3953] = {X 506.2776, Y 14.7439, Z -6.3333, A 0.000, B 0.000, C 0.000 }
gfCNCPoint5[3954] = {X 505.7970, Y 15.4954, Z -6.3333, A 0.000, B 0.000, C 0.000 }
gfCNCPoint5[3955] = {X 505.1618, Y 16.1217, Z -6.3333, A 0.000, B 0.000, C 0.000 }
gfCNCPoint5[3956] = {X 505.1617, Y 41.0652, Z -6.3333, A 0.000, B 0.000, C 0.000 }
gfCNCPoint5[3957] = {X 505.3005, Y 41.1794, Z -6.3333, A 0.000, B 0.000, C 0.000 }
gfCNCPoint5[3958] = {X 505.8863, Y 41.8058, Z -6.3333, A 0.000, B 0.000, C 0.000 }
gfCNCPoint5[3959] = {X 506.3250, Y 42.5427, Z -6.3333, A 0.000, B 0.000, C 0.000 }
gfCNCPoint5[3960] = {X 506.5966, Y 43.3562, Z -6.3333, A 0.000, B 0.000, C 0.000 }
gfCNCPoint5[3961] = {X 506.6885, Y 44.2089, Z -6.3333, A 0.000, B 0.000, C 0.000 }
gfCNCPoint5[3962] = {X 506.6885, Y 45.0000, Z -6.3333, A 0.000, B 0.000, C 0.000 }
gfCNCPoint5[3963] = {X 506.5882, Y 45.8901, Z -6.3333, A 0.000, B 0.000, C 0.000 }
gfCNCPoint5[3964] = {X 506.2924, Y 46.7355, Z -6.3333, A 0.000, B 0.000, C 0.000 }
gfCNCPoint5[3965] = {X 505.8158, Y 47.4940, Z -6.3333, A 0.000, B 0.000, C 0.000 }
gfCNCPoint5[3966] = {X 505.1825, Y 48.1273, Z -6.3333, A 0.000, B 0.000, C 0.000 }
gfCNCPoint5[3967] = {X 504.4240, Y 48.6039, Z -6.3333, A 0.000, B 0.000, C 0.000 }
gfCNCPoint5[3968] = {X 503.5786, Y 48.8997, Z -6.3333, A 0.000, B 0.000, C 0.000 }
gfCNCPoint5[3969] = {X 502.6885, Y 49.0000, Z -6.3333, A 0.000, B 0.000, C 0.000 }
gfCNCPoint5[3970] = {X 496.2450, Y 49.0000, Z -6.3333, A 0.000, B 0.000, C 0.000 }
gfCNCPoint5[3971] = {X 495.3549, Y 48.8997, Z -6.3333, A 0.000, B 0.000, C 0.000 }
gfCNCPoint5[3972] = {X 494.5095, Y 48.6039, Z -6.3333, A 0.000, B 0.000, C 0.000 }
gfCNCPoint5[3973] = {X 493.7511, Y 48.1273, Z -6.3333, A 0.000, B 0.000, C 0.000 }
gfCNCPoint5[3974] = {X 493.1177, Y 47.4939, Z -6.3333, A 0.000, B 0.000, C 0.000 }
gfCNCPoint5[3975] = {X 492.6411, Y 46.7355, Z -6.3333, A 0.000, B 0.000, C 0.000 }
gfCNCPoint5[3976] = {X 492.3453, Y 45.8901, Z -6.3333, A 0.000, B 0.000, C 0.000 }
gfCNCPoint5[3977] = {X 492.2450, Y 45.0000, Z -6.3333, A 0.000, B 0.000, C 0.000 }
gfCNCPoint5[3978] = {X 492.2454, Y 44.1538, Z -6.3333, A 0.000, B 0.000, C 0.000 }
gfCNCPoint5[3979] = {X 492.3560, Y 43.2730, Z -6.3333, A 0.000, B 0.000, C 0.000 }
gfCNCPoint5[3980] = {X 492.6582, Y 42.4382, Z -6.3333, A 0.000, B 0.000, C 0.000 }
gfCNCPoint5[3981] = {X 493.1371, Y 41.6907, Z -6.3333, A 0.000, B 0.000, C 0.000 }
gfCNCPoint5[3982] = {X 493.7690, Y 41.0672, Z -6.3333, A 0.000, B 0.000, C 0.000 }
gfCNCPoint5[3983] = {X 493.7690, Y 34.1538, Z -6.3333, A 0.000, B 0.000, C 0.000 }
gfCNCPoint5[3984] = {X 490.7739, Y 34.1538, Z -6.3333, A 0.000, B 0.000, C 0.000 }
gfCNCPoint5[3985] = {X 490.5306, Y 34.1522, Z -6.3333, A 0.000, B 0.000, C 0.000 }
gfCNCPoint5[3986] = {X 486.0915, Y 42.7966, Z -6.3333, A 0.000, B 0.000, C 0.000 }
gfCNCPoint5[3987] = {X 486.1476, Y 42.9495, Z -6.3333, A 0.000, B 0.000, C 0.000 }
gfCNCPoint5[3988] = {X 486.2998, Y 43.5710, Z -6.3333, A 0.000, B 0.000, C 0.000 }
gfCNCPoint5[3989] = {X 486.3510, Y 44.2089, Z -6.3333, A 0.000, B 0.000, C 0.000 }
gfCNCPoint5[3990] = {X 486.3510, Y 45.0000, Z -6.3333, A 0.000, B 0.000, C 0.000 }
gfCNCPoint5[3991] = {X 486.2507, Y 45.8901, Z -6.3333, A 0.000, B 0.000, C 0.000 }
gfCNCPoint5[3992] = {X 485.9549, Y 46.7355, Z -6.3333, A 0.000, B 0.000, C 0.000 }
gfCNCPoint5[3993] = {X 485.4783, Y 47.4940, Z -6.3333, A 0.000, B 0.000, C 0.000 }
gfCNCPoint5[3994] = {X 484.8450, Y 48.1273, Z -6.3333, A 0.000, B 0.000, C 0.000 }
gfCNCPoint5[3995] = {X 484.0866, Y 48.6039, Z -6.3333, A 0.000, B 0.000, C 0.000 }
gfCNCPoint5[3996] = {X 483.2411, Y 48.8997, Z -6.3333, A 0.000, B 0.000, C 0.000 }
gfCNCPoint5[3997] = {X 482.3510, Y 49.0000, Z -6.3333, A 0.000, B 0.000, C 0.000 }
gfCNCPoint5[3998] = {X 475.7650, Y 49.0000, Z -6.3333, A 0.000, B 0.000, C 0.000 }
gfCNCPoint5[3999] = {X 474.8749, Y 48.8997, Z -6.3333, A 0.000, B 0.000, C 0.000 }
gfCNCPoint5[4000] = {X 474.0294, Y 48.6039, Z -6.3333, A 0.000, B 0.000, C 0.000 }
gfCNCPoint5[4001] = {X 473.2710, Y 48.1273, Z -6.3333, A 0.000, B 0.000, C 0.000 }
gfCNCPoint5[4002] = {X 472.6376, Y 47.4940, Z -6.3333, A 0.000, B 0.000, C 0.000 }
gfCNCPoint5[4003] = {X 472.1611, Y 46.7355, Z -6.3333, A 0.000, B 0.000, C 0.000 }
gfCNCPoint5[4004] = {X 471.8652, Y 45.8901, Z -6.3333, A 0.000, B 0.000, C 0.000 }
gfCNCPoint5[4005] = {X 471.7650, Y 45.0000, Z -6.3333, A 0.000, B 0.000, C 0.000 }
gfCNCPoint5[4006] = {X 471.7653, Y 44.1538, Z -6.3333, A 0.000, B 0.000, C 0.000 }
gfCNCPoint5[4007] = {X 471.8601, Y 43.3414, Z -6.3333, A 0.000, B 0.000, C 0.000 }
gfCNCPoint5[4008] = {X 472.1182, Y 42.5654, Z -6.3333, A 0.000, B 0.000, C 0.000 }
gfCNCPoint5[4009] = {X 472.5286, Y 41.8580, Z -6.3333, A 0.000, B 0.000, C 0.000 }
gfCNCPoint5[4010] = {X 473.0744, Y 41.2489, Z -6.3333, A 0.000, B 0.000, C 0.000 }
gfCNCPoint5[4011] = {X 473.7327, Y 40.7635, Z -6.3333, A 0.000, B 0.000, C 0.000 }
gfCNCPoint5[4012] = {X 474.4759, Y 40.4222, Z -6.3333, A 0.000, B 0.000, C 0.000 }
gfCNCPoint5[4013] = {X 478.6566, Y 32.2388, Z -6.3333, A 0.000, B 0.000, C 0.000 }
gfCNCPoint5[4014] = {X 477.3654, Y 31.3993, Z -6.3333, A 0.000, B 0.000, C 0.000 }
gfCNCPoint5[4015] = {X 476.2023, Y 30.3897, Z -6.3333, A 0.000, B 0.000, C 0.000 }
gfCNCPoint5[4016] = {X 475.1898, Y 29.2292, Z -6.3333, A 0.000, B 0.000, C 0.000 }
gfCNCPoint5[4017] = {X 474.3470, Y 27.9400, Z -6.3333, A 0.000, B 0.000, C 0.000 }
gfCNCPoint5[4018] = {X 473.6902, Y 26.5470, Z -6.3333, A 0.000, B 0.000, C 0.000 }
gfCNCPoint5[4019] = {X 473.2320, Y 25.0766, Z -6.3333, A 0.000, B 0.000, C 0.000 }
gfCNCPoint5[4020] = {X 472.9240, Y 23.4256, Z -6.3333, A 0.000, B 0.000, C 0.000 }
gfCNCPoint5[4021] = {X 472.7864, Y 21.7518, Z -6.3333, A 0.000, B 0.000, C 0.000 }
gfCNCPoint5[4022] = {X 472.8204, Y 20.0727, Z -6.3333, A 0.000, B 0.000, C 0.000 }
gfCNCPoint5[4023] = {X 473.0258, Y 18.4059, Z -6.3333, A 0.000, B 0.000, C 0.000 }
gfCNCPoint5[4024] = {X 473.4004, Y 16.7687, Z -6.3333, A 0.000, B 0.000, C 0.000 }
gfCNCPoint5[4025] = {X 473.9286, Y 15.2948, Z -6.3333, A 0.000, B 0.000, C 0.000 }
gfCNCPoint5[4026] = {X 474.6519, Y 13.9061, Z -6.3333, A 0.000, B 0.000, C 0.000 }
gfCNCPoint5[4027] = {X 475.5569, Y 12.6285, Z -6.3333, A 0.000, B 0.000, C 0.000 }
gfCNCPoint5[4028] = {X 476.6269, Y 11.4854, Z -6.3333, A 0.000, B 0.000, C 0.000 }
gfCNCPoint5[4029] = {X 477.8421, Y 10.4981, Z -6.3333, A 0.000, B 0.000, C 0.000 }
gfCNCPoint5[4030] = {X 479.1801, Y 9.6848, Z -6.3333, A 0.000, B 0.000, C 0.000 }
gfCNCPoint5[4031] = {X 480.6160, Y 9.0605, Z -6.3333, A 0.000, B 0.000, C 0.000 }
gfCNCPoint5[4032] = {X 482.1233, Y 8.6368, Z -6.3333, A 0.000, B 0.000, C 0.000 }
gfCNCPoint5[4033] = {X 484.1898, Y 8.3151, Z -6.3333, A 0.000, B 0.000, C 0.000 }
gfCNCPoint5[4034] = {X 486.2782, Y 8.2021, Z -6.3333, A 0.000, B 0.000, C 0.000 }
gfCNCPoint5[4035] = {X 486.9707, Y 8.1899, Z -6.3333, A 0.000, B 0.000, C 0.000 }
gfCNCPoint5[4036] = {X 492.3835, Y 8.1899, Z -6.3333, A 0.000, B 0.000, C 0.000 }
gfCNCPoint5[4037] = {X 492.3835, Y 4.1099, Z -6.3333, A 0.000, B 0.000, C 0.000 }
gfCNCPoint5[4038] = {X 492.3835, Y 4.1099, Z -3.3333, A 0.000, B 0.000, C 0.000 }
gfCNCPoint5[4039] = {X 492.3835, Y 4.1099, Z 11.0000, A 0.000, B 0.000, C 0.000 }
gfCNCPoint5[4040] = {X 533.9635, Y 3.7897, Z 11.0000, A 0.000, B 0.000, C 0.000 }
gfCNCPoint5[4041] = {X 533.9635, Y 3.7897, Z -3.3333, A 0.000, B 0.000, C 0.000 }
gfCNCPoint5[4042] = {X 533.9635, Y 3.7897, Z -6.3333, A 0.000, B 0.000, C 0.000 }
gfCNCPoint5[4043] = {X 533.9634, Y 7.8697, Z -6.3333, A 0.000, B 0.000, C 0.000 }
gfCNCPoint5[4044] = {X 543.7499, Y 7.8699, Z -6.3333, A 0.000, B 0.000, C 0.000 }
gfCNCPoint5[4045] = {X 544.7303, Y 7.9554, Z -6.3333, A 0.000, B 0.000, C 0.000 }
gfCNCPoint5[4046] = {X 545.6659, Y 8.2603, Z -6.3333, A 0.000, B 0.000, C 0.000 }
gfCNCPoint5[4047] = {X 546.5083, Y 8.7689, Z -6.3333, A 0.000, B 0.000, C 0.000 }
gfCNCPoint5[4048] = {X 547.2140, Y 9.4547, Z -6.3333, A 0.000, B 0.000, C 0.000 }
gfCNCPoint5[4049] = {X 547.7464, Y 10.2823, Z -6.3333, A 0.000, B 0.000, C 0.000 }
gfCNCPoint5[4050] = {X 548.0779, Y 11.2089, Z -6.3333, A 0.000, B 0.000, C 0.000 }
gfCNCPoint5[4051] = {X 548.1914, Y 12.1863, Z -6.3333, A 0.000, B 0.000, C 0.000 }
gfCNCPoint5[4052] = {X 548.1912, Y 13.0225, Z -6.3333, A 0.000, B 0.000, C 0.000 }
gfCNCPoint5[4053] = {X 548.0830, Y 13.9400, Z -6.3333, A 0.000, B 0.000, C 0.000 }
gfCNCPoint5[4054] = {X 547.7821, Y 14.8135, Z -6.3333, A 0.000, B 0.000, C 0.000 }
gfCNCPoint5[4055] = {X 547.3024, Y 15.6031, Z -6.3333, A 0.000, B 0.000, C 0.000 }
gfCNCPoint5[4056] = {X 546.6658, Y 16.2726, Z -6.3333, A 0.000, B 0.000, C 0.000 }
gfCNCPoint5[4057] = {X 546.6647, Y 40.9140, Z -6.3333, A 0.000, B 0.000, C 0.000 }
gfCNCPoint5[4058] = {X 546.6865, Y 40.9320, Z -6.3333, A 0.000, B 0.000, C 0.000 }
gfCNCPoint5[4059] = {X 547.3162, Y 41.6018, Z -6.3333, A 0.000, B 0.000, C 0.000 }
gfCNCPoint5[4060] = {X 547.7898, Y 42.3897, Z -6.3333, A 0.000, B 0.000, C 0.000 }
gfCNCPoint5[4061] = {X 548.0860, Y 43.2600, Z -6.3333, A 0.000, B 0.000, C 0.000 }
gfCNCPoint5[4062] = {X 548.1913, Y 44.1733, Z -6.3333, A 0.000, B 0.000, C 0.000 }
gfCNCPoint5[4063] = {X 548.1914, Y 45.0005, Z -6.3333, A 0.000, B 0.000, C 0.000 }
gfCNCPoint5[4064] = {X 548.0779, Y 45.9779, Z -6.3333, A 0.000, B 0.000, C 0.000 }
gfCNCPoint5[4065] = {X 547.7464, Y 46.9045, Z -6.3333, A 0.000, B 0.000, C 0.000 }
gfCNCPoint5[4066] = {X 547.2140, Y 47.7320, Z -6.3333, A 0.000, B 0.000, C 0.000 }
gfCNCPoint5[4067] = {X 546.5083, Y 48.4178, Z -6.3333, A 0.000, B 0.000, C 0.000 }
gfCNCPoint5[4068] = {X 545.6658, Y 48.9263, Z -6.3333, A 0.000, B 0.000, C 0.000 }
gfCNCPoint5[4069] = {X 544.7302, Y 49.2311, Z -6.3333, A 0.000, B 0.000, C 0.000 }
gfCNCPoint5[4070] = {X 543.7499, Y 49.3166, Z -6.3333, A 0.000, B 0.000, C 0.000 }
gfCNCPoint5[4071] = {X 524.0454, Y 49.3170, Z -6.3333, A 0.000, B 0.000, C 0.000 }
gfCNCPoint5[4072] = {X 523.4988, Y 49.9508, Z -6.3333, A 0.000, B 0.000, C 0.000 }
gfCNCPoint5[4073] = {X 522.8437, Y 50.4719, Z -6.3333, A 0.000, B 0.000, C 0.000 }
gfCNCPoint5[4074] = {X 522.1031, Y 50.8619, Z -6.3333, A 0.000, B 0.000, C 0.000 }
gfCNCPoint5[4075] = {X 521.3028, Y 51.1071, Z -6.3333, A 0.000, B 0.000, C 0.000 }
gfCNCPoint5[4076] = {X 520.4708, Y 51.1991, Z -6.3333, A 0.000, B 0.000, C 0.000 }
gfCNCPoint5[4077] = {X 519.7998, Y 51.1991, Z -6.3333, A 0.000, B 0.000, C 0.000 }
gfCNCPoint5[4078] = {X 518.8385, Y 51.0908, Z -6.3333, A 0.000, B 0.000, C 0.000 }
gfCNCPoint5[4079] = {X 517.9254, Y 50.7713, Z -6.3333, A 0.000, B 0.000, C 0.000 }
gfCNCPoint5[4080] = {X 517.1063, Y 50.2566, Z -6.3333, A 0.000, B 0.000, C 0.000 }
gfCNCPoint5[4081] = {X 516.4223, Y 49.5726, Z -6.3333, A 0.000, B 0.000, C 0.000 }
gfCNCPoint5[4082] = {X 515.9076, Y 48.7535, Z -6.3333, A 0.000, B 0.000, C 0.000 }
gfCNCPoint5[4083] = {X 515.5881, Y 47.8404, Z -6.3333, A 0.000, B 0.000, C 0.000 }
gfCNCPoint5[4084] = {X 515.4798, Y 46.8791, Z -6.3333, A 0.000, B 0.000, C 0.000 }
gfCNCPoint5[4085] = {X 515.4798, Y 39.9011, Z -6.3333, A 0.000, B 0.000, C 0.000 }
gfCNCPoint5[4086] = {X 515.5869, Y 38.9451, Z -6.3333, A 0.000, B 0.000, C 0.000 }
gfCNCPoint5[4087] = {X 515.9029, Y 38.0365, Z -6.3333, A 0.000, B 0.000, C 0.000 }
gfCNCPoint5[4088] = {X 516.4121, Y 37.2204, Z -6.3333, A 0.000, B 0.000, C 0.000 }
gfCNCPoint5[4089] = {X 517.0893, Y 36.5372, Z -6.3333, A 0.000, B 0.000, C 0.000 }
gfCNCPoint5[4090] = {X 517.9010, Y 36.0208, Z -6.3333, A 0.000, B 0.000, C 0.000 }
gfCNCPoint5[4091] = {X 518.8067, Y 35.6968, Z -6.3333, A 0.000, B 0.000, C 0.000 }
gfCNCPoint5[4092] = {X 519.7617, Y 35.5813, Z -6.3333, A 0.000, B 0.000, C 0.000 }
gfCNCPoint5[4093] = {X 520.5269, Y 35.5815, Z -6.3333, A 0.000, B 0.000, C 0.000 }
gfCNCPoint5[4094] = {X 521.3532, Y 35.6727, Z -6.3333, A 0.000, B 0.000, C 0.000 }
gfCNCPoint5[4095] = {X 522.1467, Y 35.9205, Z -6.3333, A 0.000, B 0.000, C 0.000 }
gfCNCPoint5[4096] = {X 522.8781, Y 36.3158, Z -6.3333, A 0.000, B 0.000, C 0.000 }
gfCNCPoint5[4097] = {X 523.5203, Y 36.8438, Z -6.3333, A 0.000, B 0.000, C 0.000 }
gfCNCPoint5[4098] = {X 524.0494, Y 37.4850, Z -6.3333, A 0.000, B 0.000, C 0.000 }
gfCNCPoint5[4099] = {X 534.6319, Y 37.4854, Z -6.3333, A 0.000, B 0.000, C 0.000 }
gfCNCPoint5[4100] = {X 534.6319, Y 33.9660, Z -6.3333, A 0.000, B 0.000, C 0.000 }
gfCNCPoint5[4101] = {X 530.1085, Y 33.9672, Z -6.3333, A 0.000, B 0.000, C 0.000 }
gfCNCPoint5[4102] = {X 529.5763, Y 34.6110, Z -6.3333, A 0.000, B 0.000, C 0.000 }
gfCNCPoint5[4103] = {X 528.9301, Y 35.1403, Z -6.3333, A 0.000, B 0.000, C 0.000 }
gfCNCPoint5[4104] = {X 528.1942, Y 35.5354, Z -6.3333, A 0.000, B 0.000, C 0.000 }
gfCNCPoint5[4105] = {X 527.3961, Y 35.7814, Z -6.3333, A 0.000, B 0.000, C 0.000 }
gfCNCPoint5[4106] = {X 526.5655, Y 35.8693, Z -6.3333, A 0.000, B 0.000, C 0.000 }
gfCNCPoint5[4107] = {X 525.8868, Y 35.8694, Z -6.3333, A 0.000, B 0.000, C 0.000 }
gfCNCPoint5[4108] = {X 524.9255, Y 35.7611, Z -6.3333, A 0.000, B 0.000, C 0.000 }
gfCNCPoint5[4109] = {X 524.0124, Y 35.4416, Z -6.3333, A 0.000, B 0.000, C 0.000 }
gfCNCPoint5[4110] = {X 523.1933, Y 34.9270, Z -6.3333, A 0.000, B 0.000, C 0.000 }
gfCNCPoint5[4111] = {X 522.5092, Y 34.2429, Z -6.3333, A 0.000, B 0.000, C 0.000 }
gfCNCPoint5[4112] = {X 521.9946, Y 33.4238, Z -6.3333, A 0.000, B 0.000, C 0.000 }
gfCNCPoint5[4113] = {X 521.6751, Y 32.5107, Z -6.3333, A 0.000, B 0.000, C 0.000 }
gfCNCPoint5[4114] = {X 521.5668, Y 31.5494, Z -6.3333, A 0.000, B 0.000, C 0.000 }
gfCNCPoint5[4115] = {X 521.5668, Y 24.5714, Z -6.3333, A 0.000, B 0.000, C 0.000 }
gfCNCPoint5[4116] = {X 521.6739, Y 23.6153, Z -6.3333, A 0.000, B 0.000, C 0.000 }
gfCNCPoint5[4117] = {X 521.9900, Y 22.7066, Z -6.3333, A 0.000, B 0.000, C 0.000 }
gfCNCPoint5[4118] = {X 522.4994, Y 21.8904, Z -6.3333, A 0.000, B 0.000, C 0.000 }
gfCNCPoint5[4119] = {X 523.1768, Y 21.2071, Z -6.3333, A 0.000, B 0.000, C 0.000 }
gfCNCPoint5[4120] = {X 523.9886, Y 20.6908, Z -6.3333, A 0.000, B 0.000, C 0.000 }
gfCNCPoint5[4121] = {X 524.8946, Y 20.3669, Z -6.3333, A 0.000, B 0.000, C 0.000 }
gfCNCPoint5[4122] = {X 525.8498, Y 20.2516, Z -6.3333, A 0.000, B 0.000, C 0.000 }
gfCNCPoint5[4123] = {X 526.5695, Y 20.2516, Z -6.3333, A 0.000, B 0.000, C 0.000 }
gfCNCPoint5[4124] = {X 527.3944, Y 20.3391, Z -6.3333, A 0.000, B 0.000, C 0.000 }
gfCNCPoint5[4125] = {X 528.1874, Y 20.5826, Z -6.3333, A 0.000, B 0.000, C 0.000 }
gfCNCPoint5[4126] = {X 528.9192, Y 20.9733, Z -6.3333, A 0.000, B 0.000, C 0.000 }
gfCNCPoint5[4127] = {X 529.5628, Y 21.4966, Z -6.3333, A 0.000, B 0.000, C 0.000 }
gfCNCPoint5[4128] = {X 530.0946, Y 22.1332, Z -6.3333, A 0.000, B 0.000, C 0.000 }
gfCNCPoint5[4129] = {X 534.6319, Y 22.1334, Z -6.3333, A 0.000, B 0.000, C 0.000 }
gfCNCPoint5[4130] = {X 534.6319, Y 19.7024, Z -6.3333, A 0.000, B 0.000, C 0.000 }
gfCNCPoint5[4131] = {X 524.1917, Y 19.7022, Z -6.3333, A 0.000, B 0.000, C 0.000 }
gfCNCPoint5[4132] = {X 523.6593, Y 20.3466, Z -6.3333, A 0.000, B 0.000, C 0.000 }
gfCNCPoint5[4133] = {X 523.0127, Y 20.8764, Z -6.3333, A 0.000, B 0.000, C 0.000 }
gfCNCPoint5[4134] = {X 522.2762, Y 21.2718, Z -6.3333, A 0.000, B 0.000, C 0.000 }
gfCNCPoint5[4135] = {X 521.4773, Y 21.5179, Z -6.3333, A 0.000, B 0.000, C 0.000 }
gfCNCPoint5[4136] = {X 520.6460, Y 21.6056, Z -6.3333, A 0.000, B 0.000, C 0.000 }
gfCNCPoint5[4137] = {X 519.9689, Y 21.6057, Z -6.3333, A 0.000, B 0.000, C 0.000 }
gfCNCPoint5[4138] = {X 519.0076, Y 21.4974, Z -6.3333, A 0.000, B 0.000, C 0.000 }
gfCNCPoint5[4139] = {X 518.0946, Y 21.1778, Z -6.3333, A 0.000, B 0.000, C 0.000 }
gfCNCPoint5[4140] = {X 517.2755, Y 20.6631, Z -6.3333, A 0.000, B 0.000, C 0.000 }
gfCNCPoint5[4141] = {X 516.5915, Y 19.9791, Z -6.3333, A 0.000, B 0.000, C 0.000 }
gfCNCPoint5[4142] = {X 516.0769, Y 19.1600, Z -6.3333, A 0.000, B 0.000, C 0.000 }
gfCNCPoint5[4143] = {X 515.7574, Y 18.2470, Z -6.3333, A 0.000, B 0.000, C 0.000 }
gfCNCPoint5[4144] = {X 515.6491, Y 17.2857, Z -6.3333, A 0.000, B 0.000, C 0.000 }
gfCNCPoint5[4145] = {X 515.6491, Y 10.3077, Z -6.3333, A 0.000, B 0.000, C 0.000 }
gfCNCPoint5[4146] = {X 515.7562, Y 9.3519, Z -6.3333, A 0.000, B 0.000, C 0.000 }
gfCNCPoint5[4147] = {X 516.0720, Y 8.4435, Z -6.3333, A 0.000, B 0.000, C 0.000 }
gfCNCPoint5[4148] = {X 516.5811, Y 7.6275, Z -6.3333, A 0.000, B 0.000, C 0.000 }
gfCNCPoint5[4149] = {X 517.2580, Y 6.9443, Z -6.3333, A 0.000, B 0.000, C 0.000 }
gfCNCPoint5[4150] = {X 518.0693, Y 6.4278, Z -6.3333, A 0.000, B 0.000, C 0.000 }
gfCNCPoint5[4151] = {X 518.9748, Y 6.1037, Z -6.3333, A 0.000, B 0.000, C 0.000 }
gfCNCPoint5[4152] = {X 519.9296, Y 5.9879, Z -6.3333, A 0.000, B 0.000, C 0.000 }
gfCNCPoint5[4153] = {X 520.6502, Y 5.9879, Z -6.3333, A 0.000, B 0.000, C 0.000 }
gfCNCPoint5[4154] = {X 521.4754, Y 6.0751, Z -6.3333, A 0.000, B 0.000, C 0.000 }
gfCNCPoint5[4155] = {X 522.2688, Y 6.3185, Z -6.3333, A 0.000, B 0.000, C 0.000 }
gfCNCPoint5[4156] = {X 523.0010, Y 6.7092, Z -6.3333, A 0.000, B 0.000, C 0.000 }
gfCNCPoint5[4157] = {X 523.6450, Y 7.2326, Z -6.3333, A 0.000, B 0.000, C 0.000 }
gfCNCPoint5[4158] = {X 524.1770, Y 7.8695, Z -6.3333, A 0.000, B 0.000, C 0.000 }
gfCNCPoint5[4159] = {X 533.9634, Y 7.8697, Z -6.3333, A 0.000, B 0.000, C 0.000 }
gfCNCPoint5[4160] = {X 533.9635, Y 3.8697, Z -6.3333, A 0.000, B 0.000, C 0.000 }
gfCNCPoint5[4161] = {X 533.9634, Y 7.9497, Z -6.3333, A 0.000, B 0.000, C 0.000 }
gfCNCPoint5[4162] = {X 543.7510, Y 7.9499, Z -6.3333, A 0.000, B 0.000, C 0.000 }
gfCNCPoint5[4163] = {X 544.7134, Y 8.0336, Z -6.3333, A 0.000, B 0.000, C 0.000 }
gfCNCPoint5[4164] = {X 545.6319, Y 8.3328, Z -6.3333, A 0.000, B 0.000, C 0.000 }
gfCNCPoint5[4165] = {X 546.4590, Y 8.8319, Z -6.3333, A 0.000, B 0.000, C 0.000 }
gfCNCPoint5[4166] = {X 547.1518, Y 9.5050, Z -6.3333, A 0.000, B 0.000, C 0.000 }
gfCNCPoint5[4167] = {X 547.6745, Y 10.3174, Z -6.3333, A 0.000, B 0.000, C 0.000 }
gfCNCPoint5[4168] = {X 548.0000, Y 11.2269, Z -6.3333, A 0.000, B 0.000, C 0.000 }
gfCNCPoint5[4169] = {X 548.1114, Y 12.1865, Z -6.3333, A 0.000, B 0.000, C 0.000 }
gfCNCPoint5[4170] = {X 548.1112, Y 13.0217, Z -6.3333, A 0.000, B 0.000, C 0.000 }
gfCNCPoint5[4171] = {X 548.0029, Y 13.9312, Z -6.3333, A 0.000, B 0.000, C 0.000 }
gfCNCPoint5[4172] = {X 547.7018, Y 14.7962, Z -6.3333, A 0.000, B 0.000, C 0.000 }
gfCNCPoint5[4173] = {X 547.2220, Y 15.5764, Z -6.3333, A 0.000, B 0.000, C 0.000 }
gfCNCPoint5[4174] = {X 546.5858, Y 16.2353, Z -6.3333, A 0.000, B 0.000, C 0.000 }
gfCNCPoint5[4175] = {X 546.5847, Y 40.9519, Z -6.3333, A 0.000, B 0.000, C 0.000 }
gfCNCPoint5[4176] = {X 546.6351, Y 40.9932, Z -6.3333, A 0.000, B 0.000, C 0.000 }
gfCNCPoint5[4177] = {X 547.2528, Y 41.6507, Z -6.3333, A 0.000, B 0.000, C 0.000 }
gfCNCPoint5[4178] = {X 547.7174, Y 42.4238, Z -6.3333, A 0.000, B 0.000, C 0.000 }
gfCNCPoint5[4179] = {X 548.0080, Y 43.2778, Z -6.3333, A 0.000, B 0.000, C 0.000 }
gfCNCPoint5[4180] = {X 548.1113, Y 44.1740, Z -6.3333, A 0.000, B 0.000, C 0.000 }
gfCNCPoint5[4181] = {X 548.1114, Y 45.0004, Z -6.3333, A 0.000, B 0.000, C 0.000 }
gfCNCPoint5[4182] = {X 548.0000, Y 45.9599, Z -6.3333, A 0.000, B 0.000, C 0.000 }
gfCNCPoint5[4183] = {X 547.6745, Y 46.8694, Z -6.3333, A 0.000, B 0.000, C 0.000 }
gfCNCPoint5[4184] = {X 547.1518, Y 47.6817, Z -6.3333, A 0.000, B 0.000, C 0.000 }
gfCNCPoint5[4185] = {X 546.4590, Y 48.3548, Z -6.3333, A 0.000, B 0.000, C 0.000 }
gfCNCPoint5[4186] = {X 545.6319, Y 48.8539, Z -6.3333, A 0.000, B 0.000, C 0.000 }
gfCNCPoint5[4187] = {X 544.7134, Y 49.1529, Z -6.3333, A 0.000, B 0.000, C 0.000 }
gfCNCPoint5[4188] = {X 543.7510, Y 49.2366, Z -6.3333, A 0.000, B 0.000, C 0.000 }
gfCNCPoint5[4189] = {X 524.0039, Y 49.2370, Z -6.3333, A 0.000, B 0.000, C 0.000 }
gfCNCPoint5[4190] = {X 523.4671, Y 49.8702, Z -6.3333, A 0.000, B 0.000, C 0.000 }
gfCNCPoint5[4191] = {X 522.8208, Y 50.3912, Z -6.3333, A 0.000, B 0.000, C 0.000 }
gfCNCPoint5[4192] = {X 522.0881, Y 50.7814, Z -6.3333, A 0.000, B 0.000, C 0.000 }
gfCNCPoint5[4193] = {X 521.2952, Y 51.0270, Z -6.3333, A 0.000, B 0.000, C 0.000 }
gfCNCPoint5[4194] = {X 520.4702, Y 51.1191, Z -6.3333, A 0.000, B 0.000, C 0.000 }
gfCNCPoint5[4195] = {X 519.7998, Y 51.1191, Z -6.3333, A 0.000, B 0.000, C 0.000 }
gfCNCPoint5[4196] = {X 518.8563, Y 51.0128, Z -6.3333, A 0.000, B 0.000, C 0.000 }
gfCNCPoint5[4197] = {X 517.9601, Y 50.6992, Z -6.3333, A 0.000, B 0.000, C 0.000 }
gfCNCPoint5[4198] = {X 517.1562, Y 50.1941, Z -6.3333, A 0.000, B 0.000, C 0.000 }
gfCNCPoint5[4199] = {X 516.4848, Y 49.5227, Z -6.3333, A 0.000, B 0.000, C 0.000 }
gfCNCPoint5[4200] = {X 515.9797, Y 48.7188, Z -6.3333, A 0.000, B 0.000, C 0.000 }
gfCNCPoint5[4201] = {X 515.6661, Y 47.8226, Z -6.3333, A 0.000, B 0.000, C 0.000 }
gfCNCPoint5[4202] = {X 515.5598, Y 46.8791, Z -6.3333, A 0.000, B 0.000, C 0.000 }
gfCNCPoint5[4203] = {X 515.5598, Y 39.9011, Z -6.3333, A 0.000, B 0.000, C 0.000 }
gfCNCPoint5[4204] = {X 515.6649, Y 38.9628, Z -6.3333, A 0.000, B 0.000, C 0.000 }
gfCNCPoint5[4205] = {X 515.9751, Y 38.0710, Z -6.3333, A 0.000, B 0.000, C 0.000 }
gfCNCPoint5[4206] = {X 516.4749, Y 37.2700, Z -6.3333, A 0.000, B 0.000, C 0.000 }
gfCNCPoint5[4207] = {X 517.1395, Y 36.5995, Z -6.3333, A 0.000, B 0.000, C 0.000 }
gfCNCPoint5[4208] = {X 517.9361, Y 36.0926, Z -6.3333, A 0.000, B 0.000, C 0.000 }
gfCNCPoint5[4209] = {X 518.8251, Y 35.7746, Z -6.3333, A 0.000, B 0.000, C 0.000 }
gfCNCPoint5[4210] = {X 519.7624, Y 35.6613, Z -6.3333, A 0.000, B 0.000, C 0.000 }
gfCNCPoint5[4211] = {X 520.5258, Y 35.6615, Z -6.3333, A 0.000, B 0.000, C 0.000 }
gfCNCPoint5[4212] = {X 521.3451, Y 35.7528, Z -6.3333, A 0.000, B 0.000, C 0.000 }
gfCNCPoint5[4213] = {X 522.1313, Y 36.0009, Z -6.3333, A 0.000, B 0.000, C 0.000 }
gfCNCPoint5[4214] = {X 522.8546, Y 36.3964, Z -6.3333, A 0.000, B 0.000, C 0.000 }
gfCNCPoint5[4215] = {X 523.4877, Y 36.9245, Z -6.3333, A 0.000, B 0.000, C 0.000 }
gfCNCPoint5[4216] = {X 524.0066, Y 37.5650, Z -6.3333, A 0.000, B 0.000, C 0.000 }
gfCNCPoint5[4217] = {X 534.7119, Y 37.5654, Z -6.3333, A 0.000, B 0.000, C 0.000 }
gfCNCPoint5[4218] = {X 534.7119, Y 33.8860, Z -6.3333, A 0.000, B 0.000, C 0.000 }
gfCNCPoint5[4219] = {X 530.0655, Y 33.8857, Z -6.3333, A 0.000, B 0.000, C 0.000 }
gfCNCPoint5[4220] = {X 530.0416, Y 33.9234, Z -6.3333, A 0.000, B 0.000, C 0.000 }
gfCNCPoint5[4221] = {X 529.5192, Y 34.5549, Z -6.3333, A 0.000, B 0.000, C 0.000 }
gfCNCPoint5[4222] = {X 528.8851, Y 35.0742, Z -6.3333, A 0.000, B 0.000, C 0.000 }
gfCNCPoint5[4223] = {X 528.1630, Y 35.4617, Z -6.3333, A 0.000, B 0.000, C 0.000 }
gfCNCPoint5[4224] = {X 527.3798, Y 35.7031, Z -6.3333, A 0.000, B 0.000, C 0.000 }
gfCNCPoint5[4225] = {X 526.5648, Y 35.7893, Z -6.3333, A 0.000, B 0.000, C 0.000 }
gfCNCPoint5[4226] = {X 525.8868, Y 35.7894, Z -6.3333, A 0.000, B 0.000, C 0.000 }
gfCNCPoint5[4227] = {X 524.9433, Y 35.6831, Z -6.3333, A 0.000, B 0.000, C 0.000 }
gfCNCPoint5[4228] = {X 524.0471, Y 35.3696, Z -6.3333, A 0.000, B 0.000, C 0.000 }
gfCNCPoint5[4229] = {X 523.2432, Y 34.8644, Z -6.3333, A 0.000, B 0.000, C 0.000 }
gfCNCPoint5[4230] = {X 522.5718, Y 34.1930, Z -6.3333, A 0.000, B 0.000, C 0.000 }
gfCNCPoint5[4231] = {X 522.0666, Y 33.3891, Z -6.3333, A 0.000, B 0.000, C 0.000 }
gfCNCPoint5[4232] = {X 521.7531, Y 32.4929, Z -6.3333, A 0.000, B 0.000, C 0.000 }
gfCNCPoint5[4233] = {X 521.6468, Y 31.5495, Z -6.3333, A 0.000, B 0.000, C 0.000 }
gfCNCPoint5[4234] = {X 521.6468, Y 24.5714, Z -6.3333, A 0.000, B 0.000, C 0.000 }
gfCNCPoint5[4235] = {X 521.7519, Y 23.6330, Z -6.3333, A 0.000, B 0.000, C 0.000 }
gfCNCPoint5[4236] = {X 522.0622, Y 22.7411, Z -6.3333, A 0.000, B 0.000, C 0.000 }
gfCNCPoint5[4237] = {X 522.5621, Y 21.9400, Z -6.3333, A 0.000, B 0.000, C 0.000 }
gfCNCPoint5[4238] = {X 523.2270, Y 21.2694, Z -6.3333, A 0.000, B 0.000, C 0.000 }
gfCNCPoint5[4239] = {X 524.0238, Y 20.7626, Z -6.3333, A 0.000, B 0.000, C 0.000 }
gfCNCPoint5[4240] = {X 524.9130, Y 20.4448, Z -6.3333, A 0.000, B 0.000, C 0.000 }
gfCNCPoint5[4241] = {X 525.8505, Y 20.3316, Z -6.3333, A 0.000, B 0.000, C 0.000 }
gfCNCPoint5[4242] = {X 526.5687, Y 20.3316, Z -6.3333, A 0.000, B 0.000, C 0.000 }
gfCNCPoint5[4243] = {X 527.3866, Y 20.4192, Z -6.3333, A 0.000, B 0.000, C 0.000 }
gfCNCPoint5[4244] = {X 528.1722, Y 20.6630, Z -6.3333, A 0.000, B 0.000, C 0.000 }
gfCNCPoint5[4245] = {X 528.8959, Y 21.0539, Z -6.3333, A 0.000, B 0.000, C 0.000 }
gfCNCPoint5[4246] = {X 529.5305, Y 21.5772, Z -6.3333, A 0.000, B 0.000, C 0.000 }
gfCNCPoint5[4247] = {X 530.0521, Y 22.2132, Z -6.3333, A 0.000, B 0.000, C 0.000 }
gfCNCPoint5[4248] = {X 534.7119, Y 22.2134, Z -6.3333, A 0.000, B 0.000, C 0.000 }
gfCNCPoint5[4249] = {X 534.7119, Y 19.6224, Z -6.3333, A 0.000, B 0.000, C 0.000 }
gfCNCPoint5[4250] = {X 524.1487, Y 19.6222, Z -6.3333, A 0.000, B 0.000, C 0.000 }
gfCNCPoint5[4251] = {X 524.1254, Y 19.6574, Z -6.3333, A 0.000, B 0.000, C 0.000 }
gfCNCPoint5[4252] = {X 523.6028, Y 20.2899, Z -6.3333, A 0.000, B 0.000, C 0.000 }
gfCNCPoint5[4253] = {X 522.9682, Y 20.8099, Z -6.3333, A 0.000, B 0.000, C 0.000 }
gfCNCPoint5[4254] = {X 522.2453, Y 21.1980, Z -6.3333, A 0.000, B 0.000, C 0.000 }
gfCNCPoint5[4255] = {X 521.4613, Y 21.4395, Z -6.3333, A 0.000, B 0.000, C 0.000 }
gfCNCPoint5[4256] = {X 520.6453, Y 21.5256, Z -6.3333, A 0.000, B 0.000, C 0.000 }
gfCNCPoint5[4257] = {X 519.9689, Y 21.5257, Z -6.3333, A 0.000, B 0.000, C 0.000 }
gfCNCPoint5[4258] = {X 519.0254, Y 21.4194, Z -6.3333, A 0.000, B 0.000, C 0.000 }
gfCNCPoint5[4259] = {X 518.1293, Y 21.1058, Z -6.3333, A 0.000, B 0.000, C 0.000 }
gfCNCPoint5[4260] = {X 517.3254, Y 20.6006, Z -6.3333, A 0.000, B 0.000, C 0.000 }
gfCNCPoint5[4261] = {X 516.6541, Y 19.9292, Z -6.3333, A 0.000, B 0.000, C 0.000 }
gfCNCPoint5[4262] = {X 516.1490, Y 19.1253, Z -6.3333, A 0.000, B 0.000, C 0.000 }
gfCNCPoint5[4263] = {X 515.8354, Y 18.2292, Z -6.3333, A 0.000, B 0.000, C 0.000 }
gfCNCPoint5[4264] = {X 515.7291, Y 17.2857, Z -6.3333, A 0.000, B 0.000, C 0.000 }
gfCNCPoint5[4265] = {X 515.7291, Y 10.3077, Z -6.3333, A 0.000, B 0.000, C 0.000 }
gfCNCPoint5[4266] = {X 515.8342, Y 9.3696, Z -6.3333, A 0.000, B 0.000, C 0.000 }
gfCNCPoint5[4267] = {X 516.1442, Y 8.4780, Z -6.3333, A 0.000, B 0.000, C 0.000 }
gfCNCPoint5[4268] = {X 516.6438, Y 7.6771, Z -6.3333, A 0.000, B 0.000, C 0.000 }
gfCNCPoint5[4269] = {X 517.3082, Y 7.0066, Z -6.3333, A 0.000, B 0.000, C 0.000 }
gfCNCPoint5[4270] = {X 518.1045, Y 6.4997, Z -6.3333, A 0.000, B 0.000, C 0.000 }
gfCNCPoint5[4271] = {X 518.9932, Y 6.1815, Z -6.3333, A 0.000, B 0.000, C 0.000 }
gfCNCPoint5[4272] = {X 519.9303, Y 6.0679, Z -6.3333, A 0.000, B 0.000, C 0.000 }
gfCNCPoint5[4273] = {X 520.6494, Y 6.0679, Z -6.3333, A 0.000, B 0.000, C 0.000 }
gfCNCPoint5[4274] = {X 521.4677, Y 6.1552, Z -6.3333, A 0.000, B 0.000, C 0.000 }
gfCNCPoint5[4275] = {X 522.2536, Y 6.3989, Z -6.3333, A 0.000, B 0.000, C 0.000 }
gfCNCPoint5[4276] = {X 522.9777, Y 6.7898, Z -6.3333, A 0.000, B 0.000, C 0.000 }
gfCNCPoint5[4277] = {X 523.6126, Y 7.3133, Z -6.3333, A 0.000, B 0.000, C 0.000 }
gfCNCPoint5[4278] = {X 524.1345, Y 7.9495, Z -6.3333, A 0.000, B 0.000, C 0.000 }
gfCNCPoint5[4279] = {X 533.9634, Y 7.9497, Z -6.3333, A 0.000, B 0.000, C 0.000 }
gfCNCPoint5[4280] = {X 533.9635, Y 3.9497, Z -6.3333, A 0.000, B 0.000, C 0.000 }
gfCNCPoint5[4281] = {X 533.9634, Y 8.0297, Z -6.3333, A 0.000, B 0.000, C 0.000 }
gfCNCPoint5[4282] = {X 543.7521, Y 8.0299, Z -6.3333, A 0.000, B 0.000, C 0.000 }
gfCNCPoint5[4283] = {X 544.6965, Y 8.1118, Z -6.3333, A 0.000, B 0.000, C 0.000 }
gfCNCPoint5[4284] = {X 545.5979, Y 8.4052, Z -6.3333, A 0.000, B 0.000, C 0.000 }
gfCNCPoint5[4285] = {X 546.4097, Y 8.8948, Z -6.3333, A 0.000, B 0.000, C 0.000 }
gfCNCPoint5[4286] = {X 547.0896, Y 9.5553, Z -6.3333, A 0.000, B 0.000, C 0.000 }
gfCNCPoint5[4287] = {X 547.6026, Y 10.3525, Z -6.3333, A 0.000, B 0.000, C 0.000 }
gfCNCPoint5[4288] = {X 547.9221, Y 11.2450, Z -6.3333, A 0.000, B 0.000, C 0.000 }
gfCNCPoint5[4289] = {X 548.0314, Y 12.1866, Z -6.3333, A 0.000, B 0.000, C 0.000 }
gfCNCPoint5[4290] = {X 548.0312, Y 13.0208, Z -6.3333, A 0.000, B 0.000, C 0.000 }
gfCNCPoint5[4291] = {X 547.9228, Y 13.9223, Z -6.3333, A 0.000, B 0.000, C 0.000 }
gfCNCPoint5[4292] = {X 547.6215, Y 14.7787, Z -6.3333, A 0.000, B 0.000, C 0.000 }
gfCNCPoint5[4293] = {X 547.1415, Y 15.5494, Z -6.3333, A 0.000, B 0.000, C 0.000 }
gfCNCPoint5[4294] = {X 546.5058, Y 16.1976, Z -6.3333, A 0.000, B 0.000, C 0.000 }
gfCNCPoint5[4295] = {X 546.5047, Y 40.9898, Z -6.3333, A 0.000, B 0.000, C 0.000 }
gfCNCPoint5[4296] = {X 546.5837, Y 41.0545, Z -6.3333, A 0.000, B 0.000, C 0.000 }
gfCNCPoint5[4297] = {X 547.1894, Y 41.6995, Z -6.3333, A 0.000, B 0.000, C 0.000 }
gfCNCPoint5[4298] = {X 547.6450, Y 42.4579, Z -6.3333, A 0.000, B 0.000, C 0.000 }
gfCNCPoint5[4299] = {X 547.9300, Y 43.2956, Z -6.3333, A 0.000, B 0.000, C 0.000 }
gfCNCPoint5[4300] = {X 548.0313, Y 44.1746, Z -6.3333, A 0.000, B 0.000, C 0.000 }
gfCNCPoint5[4301] = {X 548.0314, Y 45.0002, Z -6.3333, A 0.000, B 0.000, C 0.000 }
gfCNCPoint5[4302] = {X 547.9221, Y 45.9418, Z -6.3333, A 0.000, B 0.000, C 0.000 }
gfCNCPoint5[4303] = {X 547.6026, Y 46.8343, Z -6.3333, A 0.000, B 0.000, C 0.000 }
gfCNCPoint5[4304] = {X 547.0896, Y 47.6314, Z -6.3333, A 0.000, B 0.000, C 0.000 }
gfCNCPoint5[4305] = {X 546.4096, Y 48.2919, Z -6.3333, A 0.000, B 0.000, C 0.000 }
gfCNCPoint5[4306] = {X 545.5979, Y 48.7814, Z -6.3333, A 0.000, B 0.000, C 0.000 }
gfCNCPoint5[4307] = {X 544.6965, Y 49.0747, Z -6.3333, A 0.000, B 0.000, C 0.000 }
gfCNCPoint5[4308] = {X 543.7521, Y 49.1566, Z -6.3333, A 0.000, B 0.000, C 0.000 }
gfCNCPoint5[4309] = {X 523.9619, Y 49.1570, Z -6.3333, A 0.000, B 0.000, C 0.000 }
gfCNCPoint5[4310] = {X 523.4351, Y 49.7895, Z -6.3333, A 0.000, B 0.000, C 0.000 }
gfCNCPoint5[4311] = {X 522.7977, Y 50.3105, Z -6.3333, A 0.000, B 0.000, C 0.000 }
gfCNCPoint5[4312] = {X 522.0731, Y 50.7010, Z -6.3333, A 0.000, B 0.000, C 0.000 }
gfCNCPoint5[4313] = {X 521.2875, Y 50.9469, Z -6.3333, A 0.000, B 0.000, C 0.000 }
gfCNCPoint5[4314] = {X 520.4695, Y 51.0391, Z -6.3333, A 0.000, B 0.000, C 0.000 }
gfCNCPoint5[4315] = {X 519.7998, Y 51.0391, Z -6.3333, A 0.000, B 0.000, C 0.000 }
gfCNCPoint5[4316] = {X 518.8741, Y 50.9348, Z -6.3333, A 0.000, B 0.000, C 0.000 }
gfCNCPoint5[4317] = {X 517.9948, Y 50.6272, Z -6.3333, A 0.000, B 0.000, C 0.000 }
gfCNCPoint5[4318] = {X 517.2061, Y 50.1315, Z -6.3333, A 0.000, B 0.000, C 0.000 }
gfCNCPoint5[4319] = {X 516.5474, Y 49.4728, Z -6.3333, A 0.000, B 0.000, C 0.000 }
gfCNCPoint5[4320] = {X 516.0517, Y 48.6841, Z -6.3333, A 0.000, B 0.000, C 0.000 }
gfCNCPoint5[4321] = {X 515.7441, Y 47.8048, Z -6.3333, A 0.000, B 0.000, C 0.000 }
gfCNCPoint5[4322] = {X 515.6398, Y 46.8791, Z -6.3333, A 0.000, B 0.000, C 0.000 }
gfCNCPoint5[4323] = {X 515.6398, Y 39.9011, Z -6.3333, A 0.000, B 0.000, C 0.000 }
gfCNCPoint5[4324] = {X 515.7429, Y 38.9805, Z -6.3333, A 0.000, B 0.000, C 0.000 }
gfCNCPoint5[4325] = {X 516.0472, Y 38.1056, Z -6.3333, A 0.000, B 0.000, C 0.000 }
gfCNCPoint5[4326] = {X 516.5376, Y 37.3197, Z -6.3333, A 0.000, B 0.000, C 0.000 }
gfCNCPoint5[4327] = {X 517.1897, Y 36.6618, Z -6.3333, A 0.000, B 0.000, C 0.000 }
gfCNCPoint5[4328] = {X 517.9713, Y 36.1645, Z -6.3333, A 0.000, B 0.000, C 0.000 }
gfCNCPoint5[4329] = {X 518.8435, Y 35.8525, Z -6.3333, A 0.000, B 0.000, C 0.000 }
gfCNCPoint5[4330] = {X 519.7631, Y 35.7413, Z -6.3333, A 0.000, B 0.000, C 0.000 }
gfCNCPoint5[4331] = {X 520.5247, Y 35.7415, Z -6.3333, A 0.000, B 0.000, C 0.000 }
gfCNCPoint5[4332] = {X 521.3370, Y 35.8328, Z -6.3333, A 0.000, B 0.000, C 0.000 }
gfCNCPoint5[4333] = {X 522.1157, Y 36.0812, Z -6.3333, A 0.000, B 0.000, C 0.000 }
gfCNCPoint5[4334] = {X 522.8308, Y 36.4771, Z -6.3333, A 0.000, B 0.000, C 0.000 }
gfCNCPoint5[4335] = {X 523.4547, Y 37.0052, Z -6.3333, A 0.000, B 0.000, C 0.000 }
gfCNCPoint5[4336] = {X 523.9633, Y 37.6450, Z -6.3333, A 0.000, B 0.000, C 0.000 }
gfCNCPoint5[4337] = {X 534.7919, Y 37.6454, Z -6.3333, A 0.000, B 0.000, C 0.000 }
gfCNCPoint5[4338] = {X 534.7919, Y 33.8060, Z -6.3333, A 0.000, B 0.000, C 0.000 }
gfCNCPoint5[4339] = {X 530.0216, Y 33.8057, Z -6.3333, A 0.000, B 0.000, C 0.000 }
gfCNCPoint5[4340] = {X 529.9746, Y 33.8795, Z -6.3333, A 0.000, B 0.000, C 0.000 }
gfCNCPoint5[4341] = {X 529.4621, Y 34.4988, Z -6.3333, A 0.000, B 0.000, C 0.000 }
gfCNCPoint5[4342] = {X 528.8401, Y 35.0080, Z -6.3333, A 0.000, B 0.000, C 0.000 }
gfCNCPoint5[4343] = {X 528.1317, Y 35.3881, Z -6.3333, A 0.000, B 0.000, C 0.000 }
gfCNCPoint5[4344] = {X 527.3635, Y 35.6248, Z -6.3333, A 0.000, B 0.000, C 0.000 }
gfCNCPoint5[4345] = {X 526.5641, Y 35.7093, Z -6.3333, A 0.000, B 0.000, C 0.000 }
gfCNCPoint5[4346] = {X 525.8868, Y 35.7095, Z -6.3333, A 0.000, B 0.000, C 0.000 }
gfCNCPoint5[4347] = {X 524.9611, Y 35.6052, Z -6.3333, A 0.000, B 0.000, C 0.000 }
gfCNCPoint5[4348] = {X 524.0818, Y 35.2975, Z -6.3333, A 0.000, B 0.000, C 0.000 }
gfCNCPoint5[4349] = {X 523.2930, Y 34.8019, Z -6.3333, A 0.000, B 0.000, C 0.000 }
gfCNCPoint5[4350] = {X 522.6343, Y 34.1432, Z -6.3333, A 0.000, B 0.000, C 0.000 }
gfCNCPoint5[4351] = {X 522.1387, Y 33.3544, Z -6.3333, A 0.000, B 0.000, C 0.000 }
gfCNCPoint5[4352] = {X 521.8311, Y 32.4751, Z -6.3333, A 0.000, B 0.000, C 0.000 }
gfCNCPoint5[4353] = {X 521.7268, Y 31.5495, Z -6.3333, A 0.000, B 0.000, C 0.000 }
gfCNCPoint5[4354] = {X 521.7268, Y 24.5714, Z -6.3333, A 0.000, B 0.000, C 0.000 }
gfCNCPoint5[4355] = {X 521.8299, Y 23.6507, Z -6.3333, A 0.000, B 0.000, C 0.000 }
gfCNCPoint5[4356] = {X 522.1343, Y 22.7756, Z -6.3333, A 0.000, B 0.000, C 0.000 }
gfCNCPoint5[4357] = {X 522.6248, Y 21.9897, Z -6.3333, A 0.000, B 0.000, C 0.000 }
gfCNCPoint5[4358] = {X 523.2772, Y 21.3317, Z -6.3333, A 0.000, B 0.000, C 0.000 }
gfCNCPoint5[4359] = {X 524.0589, Y 20.8345, Z -6.3333, A 0.000, B 0.000, C 0.000 }
gfCNCPoint5[4360] = {X 524.9313, Y 20.5226, Z -6.3333, A 0.000, B 0.000, C 0.000 }
gfCNCPoint5[4361] = {X 525.8511, Y 20.4116, Z -6.3333, A 0.000, B 0.000, C 0.000 }
gfCNCPoint5[4362] = {X 526.5679, Y 20.4116, Z -6.3333, A 0.000, B 0.000, C 0.000 }
gfCNCPoint5[4363] = {X 527.3787, Y 20.4993, Z -6.3333, A 0.000, B 0.000, C 0.000 }
gfCNCPoint5[4364] = {X 528.1568, Y 20.7434, Z -6.3333, A 0.000, B 0.000, C 0.000 }
gfCNCPoint5[4365] = {X 528.8724, Y 21.1346, Z -6.3333, A 0.000, B 0.000, C 0.000 }
gfCNCPoint5[4366] = {X 529.4978, Y 21.6579, Z -6.3333, A 0.000, B 0.000, C 0.000 }
gfCNCPoint5[4367] = {X 530.0091, Y 22.2932, Z -6.3333, A 0.000, B 0.000, C 0.000 }
gfCNCPoint5[4368] = {X 534.7919, Y 22.2934, Z -6.3333, A 0.000, B 0.000, C 0.000 }
gfCNCPoint5[4369] = {X 534.7919, Y 19.5424, Z -6.3333, A 0.000, B 0.000, C 0.000 }
gfCNCPoint5[4370] = {X 524.1048, Y 19.5422, Z -6.3333, A 0.000, B 0.000, C 0.000 }
gfCNCPoint5[4371] = {X 524.0761, Y 19.5872, Z -6.3333, A 0.000, B 0.000, C 0.000 }
gfCNCPoint5[4372] = {X 523.5637, Y 20.2159, Z -6.3333, A 0.000, B 0.000, C 0.000 }
gfCNCPoint5[4373] = {X 522.9390, Y 20.7332, Z -6.3333, A 0.000, B 0.000, C 0.000 }
gfCNCPoint5[4374] = {X 522.2258, Y 21.1194, Z -6.3333, A 0.000, B 0.000, C 0.000 }
gfCNCPoint5[4375] = {X 521.4512, Y 21.3599, Z -6.3333, A 0.000, B 0.000, C 0.000 }
gfCNCPoint5[4376] = {X 520.6447, Y 21.4456, Z -6.3333, A 0.000, B 0.000, C 0.000 }
gfCNCPoint5[4377] = {X 519.9689, Y 21.4457, Z -6.3333, A 0.000, B 0.000, C 0.000 }
gfCNCPoint5[4378] = {X 519.0432, Y 21.3414, Z -6.3333, A 0.000, B 0.000, C 0.000 }
gfCNCPoint5[4379] = {X 518.1640, Y 21.0337, Z -6.3333, A 0.000, B 0.000, C 0.000 }
gfCNCPoint5[4380] = {X 517.3753, Y 20.5381, Z -6.3333, A 0.000, B 0.000, C 0.000 }
gfCNCPoint5[4381] = {X 516.7166, Y 19.8794, Z -6.3333, A 0.000, B 0.000, C 0.000 }
gfCNCPoint5[4382] = {X 516.2210, Y 19.0906, Z -6.3333, A 0.000, B 0.000, C 0.000 }
gfCNCPoint5[4383] = {X 515.9134, Y 18.2114, Z -6.3333, A 0.000, B 0.000, C 0.000 }
gfCNCPoint5[4384] = {X 515.8091, Y 17.2857, Z -6.3333, A 0.000, B 0.000, C 0.000 }
gfCNCPoint5[4385] = {X 515.8091, Y 10.3077, Z -6.3333, A 0.000, B 0.000, C 0.000 }
gfCNCPoint5[4386] = {X 515.9122, Y 9.3873, Z -6.3333, A 0.000, B 0.000, C 0.000 }
gfCNCPoint5[4387] = {X 516.2164, Y 8.5125, Z -6.3333, A 0.000, B 0.000, C 0.000 }
gfCNCPoint5[4388] = {X 516.7065, Y 7.7267, Z -6.3333, A 0.000, B 0.000, C 0.000 }
gfCNCPoint5[4389] = {X 517.3584, Y 7.0689, Z -6.3333, A 0.000, B 0.000, C 0.000 }
gfCNCPoint5[4390] = {X 518.1397, Y 6.5715, Z -6.3333, A 0.000, B 0.000, C 0.000 }
gfCNCPoint5[4391] = {X 519.0117, Y 6.2594, Z -6.3333, A 0.000, B 0.000, C 0.000 }
gfCNCPoint5[4392] = {X 519.9311, Y 6.1479, Z -6.3333, A 0.000, B 0.000, C 0.000 }
gfCNCPoint5[4393] = {X 520.6487, Y 6.1479, Z -6.3333, A 0.000, B 0.000, C 0.000 }
gfCNCPoint5[4394] = {X 521.4598, Y 6.2353, Z -6.3333, A 0.000, B 0.000, C 0.000 }
gfCNCPoint5[4395] = {X 522.2383, Y 6.4793, Z -6.3333, A 0.000, B 0.000, C 0.000 }
gfCNCPoint5[4396] = {X 522.9542, Y 6.8705, Z -6.3333, A 0.000, B 0.000, C 0.000 }
gfCNCPoint5[4397] = {X 523.5800, Y 7.3940, Z -6.3333, A 0.000, B 0.000, C 0.000 }
gfCNCPoint5[4398] = {X 524.0915, Y 8.0295, Z -6.3333, A 0.000, B 0.000, C 0.000 }
gfCNCPoint5[4399] = {X 533.9634, Y 8.0297, Z -6.3333, A 0.000, B 0.000, C 0.000 }
gfCNCPoint5[4400] = {X 533.9635, Y 4.0297, Z -6.3333, A 0.000, B 0.000, C 0.000 }
gfCNCPoint5[4401] = {X 533.9634, Y 8.1097, Z -6.3333, A 0.000, B 0.000, C 0.000 }
gfCNCPoint5[4402] = {X 543.7532, Y 8.1099, Z -6.3333, A 0.000, B 0.000, C 0.000 }
gfCNCPoint5[4403] = {X 544.6797, Y 8.1900, Z -6.3333, A 0.000, B 0.000, C 0.000 }
gfCNCPoint5[4404] = {X 545.5640, Y 8.4776, Z -6.3333, A 0.000, B 0.000, C 0.000 }
gfCNCPoint5[4405] = {X 546.3603, Y 8.9578, Z -6.3333, A 0.000, B 0.000, C 0.000 }
gfCNCPoint5[4406] = {X 547.0274, Y 9.6056, Z -6.3333, A 0.000, B 0.000, C 0.000 }
gfCNCPoint5[4407] = {X 547.5307, Y 10.3875, Z -6.3333, A 0.000, B 0.000, C 0.000 }
gfCNCPoint5[4408] = {X 547.8441, Y 11.2630, Z -6.3333, A 0.000, B 0.000, C 0.000 }
gfCNCPoint5[4409] = {X 547.9514, Y 12.1867, Z -6.3333, A 0.000, B 0.000, C 0.000 }
gfCNCPoint5[4410] = {X 547.9512, Y 13.0200, Z -6.3333, A 0.000, B 0.000, C 0.000 }
gfCNCPoint5[4411] = {X 547.8428, Y 13.9133, Z -6.3333, A 0.000, B 0.000, C 0.000 }
gfCNCPoint5[4412] = {X 547.5412, Y 14.7611, Z -6.3333, A 0.000, B 0.000, C 0.000 }
gfCNCPoint5[4413] = {X 547.0611, Y 15.5222, Z -6.3333, A 0.000, B 0.000, C 0.000 }
gfCNCPoint5[4414] = {X 546.4258, Y 16.1595, Z -6.3333, A 0.000, B 0.000, C 0.000 }
gfCNCPoint5[4415] = {X 546.4247, Y 41.0276, Z -6.3333, A 0.000, B 0.000, C 0.000 }
gfCNCPoint5[4416] = {X 546.5322, Y 41.1158, Z -6.3333, A 0.000, B 0.000, C 0.000 }
gfCNCPoint5[4417] = {X 547.1260, Y 41.7483, Z -6.3333, A 0.000, B 0.000, C 0.000 }
gfCNCPoint5[4418] = {X 547.5727, Y 42.4920, Z -6.3333, A 0.000, B 0.000, C 0.000 }
gfCNCPoint5[4419] = {X 547.8520, Y 43.3134, Z -6.3333, A 0.000, B 0.000, C 0.000 }
gfCNCPoint5[4420] = {X 547.9513, Y 44.1753, Z -6.3333, A 0.000, B 0.000, C 0.000 }
gfCNCPoint5[4421] = {X 547.9514, Y 45.0001, Z -6.3333, A 0.000, B 0.000, C 0.000 }
gfCNCPoint5[4422] = {X 547.8441, Y 45.9238, Z -6.3333, A 0.000, B 0.000, C 0.000 }
gfCNCPoint5[4423] = {X 547.5307, Y 46.7992, Z -6.3333, A 0.000, B 0.000, C 0.000 }
gfCNCPoint5[4424] = {X 547.0274, Y 47.5811, Z -6.3333, A 0.000, B 0.000, C 0.000 }
gfCNCPoint5[4425] = {X 546.3603, Y 48.2289, Z -6.3333, A 0.000, B 0.000, C 0.000 }
gfCNCPoint5[4426] = {X 545.5639, Y 48.7090, Z -6.3333, A 0.000, B 0.000, C 0.000 }
gfCNCPoint5[4427] = {X 544.6796, Y 48.9965, Z -6.3333, A 0.000, B 0.000, C 0.000 }
gfCNCPoint5[4428] = {X 543.7532, Y 49.0766, Z -6.3333, A 0.000, B 0.000, C 0.000 }
gfCNCPoint5[4429] = {X 523.9194, Y 49.0770, Z -6.3333, A 0.000, B 0.000, C 0.000 }
gfCNCPoint5[4430] = {X 523.4027, Y 49.7087, Z -6.3333, A 0.000, B 0.000, C 0.000 }
gfCNCPoint5[4431] = {X 522.7744, Y 50.2297, Z -6.3333, A 0.000, B 0.000, C 0.000 }
gfCNCPoint5[4432] = {X 522.0579, Y 50.6206, Z -6.3333, A 0.000, B 0.000, C 0.000 }
gfCNCPoint5[4433] = {X 521.2797, Y 50.8667, Z -6.3333, A 0.000, B 0.000, C 0.000 }
gfCNCPoint5[4434] = {X 520.4688, Y 50.9591, Z -6.3333, A 0.000, B 0.000, C 0.000 }
gfCNCPoint5[4435] = {X 519.7998, Y 50.9591, Z -6.3333, A 0.000, B 0.000, C 0.000 }
gfCNCPoint5[4436] = {X 518.8919, Y 50.8568, Z -6.3333, A 0.000, B 0.000, C 0.000 }
gfCNCPoint5[4437] = {X 518.0295, Y 50.5551, Z -6.3333, A 0.000, B 0.000, C 0.000 }
gfCNCPoint5[4438] = {X 517.2559, Y 50.0690, Z -6.3333, A 0.000, B 0.000, C 0.000 }
gfCNCPoint5[4439] = {X 516.6099, Y 49.4230, Z -6.3333, A 0.000, B 0.000, C 0.000 }
gfCNCPoint5[4440] = {X 516.1238, Y 48.6494, Z -6.3333, A 0.000, B 0.000, C 0.000 }
gfCNCPoint5[4441] = {X 515.8221, Y 47.7870, Z -6.3333, A 0.000, B 0.000, C 0.000 }
gfCNCPoint5[4442] = {X 515.7198, Y 46.8791, Z -6.3333, A 0.000, B 0.000, C 0.000 }
gfCNCPoint5[4443] = {X 515.7198, Y 39.9011, Z -6.3333, A 0.000, B 0.000, C 0.000 }
gfCNCPoint5[4444] = {X 515.8209, Y 38.9982, Z -6.3333, A 0.000, B 0.000, C 0.000 }
gfCNCPoint5[4445] = {X 516.1194, Y 38.1401, Z -6.3333, A 0.000, B 0.000, C 0.000 }
gfCNCPoint5[4446] = {X 516.6003, Y 37.3693, Z -6.3333, A 0.000, B 0.000, C 0.000 }
gfCNCPoint5[4447] = {X 517.2399, Y 36.7241, Z -6.3333, A 0.000, B 0.000, C 0.000 }
gfCNCPoint5[4448] = {X 518.0064, Y 36.2364, Z -6.3333, A 0.000, B 0.000, C 0.000 }
gfCNCPoint5[4449] = {X 518.8619, Y 35.9304, Z -6.3333, A 0.000, B 0.000, C 0.000 }
gfCNCPoint5[4450] = {X 519.7638, Y 35.8213, Z -6.3333, A 0.000, B 0.000, C 0.000 }
gfCNCPoint5[4451] = {X 520.5236, Y 35.8215, Z -6.3333, A 0.000, B 0.000, C 0.000 }
gfCNCPoint5[4452] = {X 521.3287, Y 35.9129, Z -6.3333, A 0.000, B 0.000, C 0.000 }
gfCNCPoint5[4453] = {X 522.0999, Y 36.1616, Z -6.3333, A 0.000, B 0.000, C 0.000 }
gfCNCPoint5[4454] = {X 522.8067, Y 36.5578, Z -6.3333, A 0.000, B 0.000, C 0.000 }
gfCNCPoint5[4455] = {X 523.4213, Y 37.0859, Z -6.3333, A 0.000, B 0.000, C 0.000 }
gfCNCPoint5[4456] = {X 523.9194, Y 37.7250, Z -6.3333, A 0.000, B 0.000, C 0.000 }
gfCNCPoint5[4457] = {X 534.8719, Y 37.7254, Z -6.3333, A 0.000, B 0.000, C 0.000 }
gfCNCPoint5[4458] = {X 534.8719, Y 33.7260, Z -6.3333, A 0.000, B 0.000, C 0.000 }
gfCNCPoint5[4459] = {X 529.9776, Y 33.7257, Z -6.3333, A 0.000, B 0.000, C 0.000 }
gfCNCPoint5[4460] = {X 529.9071, Y 33.8366, Z -6.3333, A 0.000, B 0.000, C 0.000 }
gfCNCPoint5[4461] = {X 529.2612, Y 34.5790, Z -6.3333, A 0.000, B 0.000, C 0.000 }
gfCNCPoint5[4462] = {X 528.4563, Y 35.1452, Z -6.3333, A 0.000, B 0.000, C 0.000 }
gfCNCPoint5[4463] = {X 527.5392, Y 35.5023, Z -6.3333, A 0.000, B 0.000, C 0.000 }
gfCNCPoint5[4464] = {X 526.5634, Y 35.6293, Z -6.3333, A 0.000, B 0.000, C 0.000 }
gfCNCPoint5[4465] = {X 525.8868, Y 35.6295, Z -6.3333, A 0.000, B 0.000, C 0.000 }
gfCNCPoint5[4466] = {X 524.9789, Y 35.5272, Z -6.3333, A 0.000, B 0.000, C 0.000 }
gfCNCPoint5[4467] = {X 524.1165, Y 35.2254, Z -6.3333, A 0.000, B 0.000, C 0.000 }
gfCNCPoint5[4468] = {X 523.3429, Y 34.7393, Z -6.3333, A 0.000, B 0.000, C 0.000 }
gfCNCPoint5[4469] = {X 522.6969, Y 34.0933, Z -6.3333, A 0.000, B 0.000, C 0.000 }
gfCNCPoint5[4470] = {X 522.2108, Y 33.3197, Z -6.3333, A 0.000, B 0.000, C 0.000 }
gfCNCPoint5[4471] = {X 521.9091, Y 32.4573, Z -6.3333, A 0.000, B 0.000, C 0.000 }
gfCNCPoint5[4472] = {X 521.8068, Y 31.5495, Z -6.3333, A 0.000, B 0.000, C 0.000 }
gfCNCPoint5[4473] = {X 521.8068, Y 24.5714, Z -6.3333, A 0.000, B 0.000, C 0.000 }
gfCNCPoint5[4474] = {X 521.9079, Y 23.6684, Z -6.3333, A 0.000, B 0.000, C 0.000 }
gfCNCPoint5[4475] = {X 522.2065, Y 22.8102, Z -6.3333, A 0.000, B 0.000, C 0.000 }
gfCNCPoint5[4476] = {X 522.6876, Y 22.0393, Z -6.3333, A 0.000, B 0.000, C 0.000 }
gfCNCPoint5[4477] = {X 523.3273, Y 21.3940, Z -6.3333, A 0.000, B 0.000, C 0.000 }
gfCNCPoint5[4478] = {X 524.0941, Y 20.9064, Z -6.3333, A 0.000, B 0.000, C 0.000 }
gfCNCPoint5[4479] = {X 524.9497, Y 20.6005, Z -6.3333, A 0.000, B 0.000, C 0.000 }
gfCNCPoint5[4480] = {X 525.8518, Y 20.4916, Z -6.3333, A 0.000, B 0.000, C 0.000 }
gfCNCPoint5[4481] = {X 526.5672, Y 20.4916, Z -6.3333, A 0.000, B 0.000, C 0.000 }
gfCNCPoint5[4482] = {X 527.3708, Y 20.5793, Z -6.3333, A 0.000, B 0.000, C 0.000 }
gfCNCPoint5[4483] = {X 528.1414, Y 20.8238, Z -6.3333, A 0.000, B 0.000, C 0.000 }
gfCNCPoint5[4484] = {X 528.8486, Y 21.2154, Z -6.3333, A 0.000, B 0.000, C 0.000 }
gfCNCPoint5[4485] = {X 529.4647, Y 21.7387, Z -6.3333, A 0.000, B 0.000, C 0.000 }
gfCNCPoint5[4486] = {X 529.9656, Y 22.3732, Z -6.3333, A 0.000, B 0.000, C 0.000 }
gfCNCPoint5[4487] = {X 534.8719, Y 22.3734, Z -6.3333, A 0.000, B 0.000, C 0.000 }
gfCNCPoint5[4488] = {X 534.8719, Y 19.4624, Z -6.3333, A 0.000, B 0.000, C 0.000 }
gfCNCPoint5[4489] = {X 524.0610, Y 19.4622, Z -6.3333, A 0.000, B 0.000, C 0.000 }
gfCNCPoint5[4490] = {X 524.0087, Y 19.5442, Z -6.3333, A 0.000, B 0.000, C 0.000 }
gfCNCPoint5[4491] = {X 523.5061, Y 20.1604, Z -6.3333, A 0.000, B 0.000, C 0.000 }
gfCNCPoint5[4492] = {X 522.8935, Y 20.6674, Z -6.3333, A 0.000, B 0.000, C 0.000 }
gfCNCPoint5[4493] = {X 522.1942, Y 21.0459, Z -6.3333, A 0.000, B 0.000, C 0.000 }
gfCNCPoint5[4494] = {X 521.4348, Y 21.2816, Z -6.3333, A 0.000, B 0.000, C 0.000 }
gfCNCPoint5[4495] = {X 520.6440, Y 21.3656, Z -6.3333, A 0.000, B 0.000, C 0.000 }
gfCNCPoint5[4496] = {X 519.9689, Y 21.3657, Z -6.3333, A 0.000, B 0.000, C 0.000 }
gfCNCPoint5[4497] = {X 519.0610, Y 21.2634, Z -6.3333, A 0.000, B 0.000, C 0.000 }
gfCNCPoint5[4498] = {X 518.1987, Y 20.9616, Z -6.3333, A 0.000, B 0.000, C 0.000 }
gfCNCPoint5[4499] = {X 517.4252, Y 20.4755, Z -6.3333, A 0.000, B 0.000, C 0.000 }
gfCNCPoint5[4500] = {X 516.7792, Y 19.8295, Z -6.3333, A 0.000, B 0.000, C 0.000 }
gfCNCPoint5[4501] = {X 516.2931, Y 19.0559, Z -6.3333, A 0.000, B 0.000, C 0.000 }
gfCNCPoint5[4502] = {X 515.9914, Y 18.1936, Z -6.3333, A 0.000, B 0.000, C 0.000 }
gfCNCPoint5[4503] = {X 515.8891, Y 17.2857, Z -6.3333, A 0.000, B 0.000, C 0.000 }
gfCNCPoint5[4504] = {X 515.8891, Y 10.3077, Z -6.3333, A 0.000, B 0.000, C 0.000 }
gfCNCPoint5[4505] = {X 515.9902, Y 9.4050, Z -6.3333, A 0.000, B 0.000, C 0.000 }
gfCNCPoint5[4506] = {X 516.2885, Y 8.5471, Z -6.3333, A 0.000, B 0.000, C 0.000 }
gfCNCPoint5[4507] = {X 516.7693, Y 7.7764, Z -6.3333, A 0.000, B 0.000, C 0.000 }
gfCNCPoint5[4508] = {X 517.4086, Y 7.1312, Z -6.3333, A 0.000, B 0.000, C 0.000 }
gfCNCPoint5[4509] = {X 518.1749, Y 6.6434, Z -6.3333, A 0.000, B 0.000, C 0.000 }
gfCNCPoint5[4510] = {X 519.0301, Y 6.3372, Z -6.3333, A 0.000, B 0.000, C 0.000 }
gfCNCPoint5[4511] = {X 519.9318, Y 6.2279, Z -6.3333, A 0.000, B 0.000, C 0.000 }
gfCNCPoint5[4512] = {X 520.6480, Y 6.2279, Z -6.3333, A 0.000, B 0.000, C 0.000 }
gfCNCPoint5[4513] = {X 521.4520, Y 6.3153, Z -6.3333, A 0.000, B 0.000, C 0.000 }
gfCNCPoint5[4514] = {X 522.2229, Y 6.5597, Z -6.3333, A 0.000, B 0.000, C 0.000 }
gfCNCPoint5[4515] = {X 522.9305, Y 6.9513, Z -6.3333, A 0.000, B 0.000, C 0.000 }
gfCNCPoint5[4516] = {X 523.5469, Y 7.4747, Z -6.3333, A 0.000, B 0.000, C 0.000 }
gfCNCPoint5[4517] = {X 524.0480, Y 8.1095, Z -6.3333, A 0.000, B 0.000, C 0.000 }
gfCNCPoint5[4518] = {X 533.9634, Y 8.1097, Z -6.3333, A 0.000, B 0.000, C 0.000 }
gfCNCPoint5[4519] = {X 533.9635, Y 4.1097, Z -6.3333, A 0.000, B 0.000, C 0.000 }
gfCNCPoint5[4520] = {X 533.9634, Y 8.1897, Z -6.3333, A 0.000, B 0.000, C 0.000 }
gfCNCPoint5[4521] = {X 543.7544, Y 8.1899, Z -6.3333, A 0.000, B 0.000, C 0.000 }
gfCNCPoint5[4522] = {X 544.6628, Y 8.2683, Z -6.3333, A 0.000, B 0.000, C 0.000 }
gfCNCPoint5[4523] = {X 545.5300, Y 8.5501, Z -6.3333, A 0.000, B 0.000, C 0.000 }
gfCNCPoint5[4524] = {X 546.3110, Y 9.0208, Z -6.3333, A 0.000, B 0.000, C 0.000 }
gfCNCPoint5[4525] = {X 546.9652, Y 9.6559, Z -6.3333, A 0.000, B 0.000, C 0.000 }
gfCNCPoint5[4526] = {X 547.4588, Y 10.4226, Z -6.3333, A 0.000, B 0.000, C 0.000 }
gfCNCPoint5[4527] = {X 547.7662, Y 11.2811, Z -6.3333, A 0.000, B 0.000, C 0.000 }
gfCNCPoint5[4528] = {X 547.8714, Y 12.1868, Z -6.3333, A 0.000, B 0.000, C 0.000 }
gfCNCPoint5[4529] = {X 547.8712, Y 13.0192, Z -6.3333, A 0.000, B 0.000, C 0.000 }
gfCNCPoint5[4530] = {X 547.7627, Y 13.9043, Z -6.3333, A 0.000, B 0.000, C 0.000 }
gfCNCPoint5[4531] = {X 547.4608, Y 14.7433, Z -6.3333, A 0.000, B 0.000, C 0.000 }
gfCNCPoint5[4532] = {X 546.9806, Y 15.4946, Z -6.3333, A 0.000, B 0.000, C 0.000 }
gfCNCPoint5[4533] = {X 546.3458, Y 16.1209, Z -6.3333, A 0.000, B 0.000, C 0.000 }
gfCNCPoint5[4534] = {X 546.3447, Y 41.0655, Z -6.3333, A 0.000, B 0.000, C 0.000 }
gfCNCPoint5[4535] = {X 546.4835, Y 41.1794, Z -6.3333, A 0.000, B 0.000, C 0.000 }
gfCNCPoint5[4536] = {X 547.0692, Y 41.8058, Z -6.3333, A 0.000, B 0.000, C 0.000 }
gfCNCPoint5[4537] = {X 547.5079, Y 42.5427, Z -6.3333, A 0.000, B 0.000, C 0.000 }
gfCNCPoint5[4538] = {X 547.7795, Y 43.3562, Z -6.3333, A 0.000, B 0.000, C 0.000 }
gfCNCPoint5[4539] = {X 547.8714, Y 44.2089, Z -6.3333, A 0.000, B 0.000, C 0.000 }
gfCNCPoint5[4540] = {X 547.8714, Y 45.0000, Z -6.3333, A 0.000, B 0.000, C 0.000 }
gfCNCPoint5[4541] = {X 547.7662, Y 45.9057, Z -6.3333, A 0.000, B 0.000, C 0.000 }
gfCNCPoint5[4542] = {X 547.4588, Y 46.7641, Z -6.3333, A 0.000, B 0.000, C 0.000 }
gfCNCPoint5[4543] = {X 546.9652, Y 47.5308, Z -6.3333, A 0.000, B 0.000, C 0.000 }
gfCNCPoint5[4544] = {X 546.3110, Y 48.1659, Z -6.3333, A 0.000, B 0.000, C 0.000 }
gfCNCPoint5[4545] = {X 545.5300, Y 48.6365, Z -6.3333, A 0.000, B 0.000, C 0.000 }
gfCNCPoint5[4546] = {X 544.6628, Y 48.9183, Z -6.3333, A 0.000, B 0.000, C 0.000 }
gfCNCPoint5[4547] = {X 543.7544, Y 48.9966, Z -6.3333, A 0.000, B 0.000, C 0.000 }
gfCNCPoint5[4548] = {X 523.8764, Y 48.9970, Z -6.3333, A 0.000, B 0.000, C 0.000 }
gfCNCPoint5[4549] = {X 523.3700, Y 49.6280, Z -6.3333, A 0.000, B 0.000, C 0.000 }
gfCNCPoint5[4550] = {X 522.7509, Y 50.1489, Z -6.3333, A 0.000, B 0.000, C 0.000 }
gfCNCPoint5[4551] = {X 522.0426, Y 50.5401, Z -6.3333, A 0.000, B 0.000, C 0.000 }
gfCNCPoint5[4552] = {X 521.2719, Y 50.7866, Z -6.3333, A 0.000, B 0.000, C 0.000 }
gfCNCPoint5[4553] = {X 520.4681, Y 50.8791, Z -6.3333, A 0.000, B 0.000, C 0.000 }
gfCNCPoint5[4554] = {X 519.7998, Y 50.8791, Z -6.3333, A 0.000, B 0.000, C 0.000 }
gfCNCPoint5[4555] = {X 518.9097, Y 50.7788, Z -6.3333, A 0.000, B 0.000, C 0.000 }
gfCNCPoint5[4556] = {X 518.0642, Y 50.4830, Z -6.3333, A 0.000, B 0.000, C 0.000 }
gfCNCPoint5[4557] = {X 517.3058, Y 50.0064, Z -6.3333, A 0.000, B 0.000, C 0.000 }
gfCNCPoint5[4558] = {X 516.6724, Y 49.3731, Z -6.3333, A 0.000, B 0.000, C 0.000 }
gfCNCPoint5[4559] = {X 516.1959, Y 48.6147, Z -6.3333, A 0.000, B 0.000, C 0.000 }
gfCNCPoint5[4560] = {X 515.9001, Y 47.7692, Z -6.3333, A 0.000, B 0.000, C 0.000 }
gfCNCPoint5[4561] = {X 515.7998, Y 46.8791, Z -6.3333, A 0.000, B 0.000, C 0.000 }
gfCNCPoint5[4562] = {X 515.7998, Y 39.9011, Z -6.3333, A 0.000, B 0.000, C 0.000 }
gfCNCPoint5[4563] = {X 515.9001, Y 39.0110, Z -6.3333, A 0.000, B 0.000, C 0.000 }
gfCNCPoint5[4564] = {X 516.1959, Y 38.1655, Z -6.3333, A 0.000, B 0.000, C 0.000 }
gfCNCPoint5[4565] = {X 516.6725, Y 37.4071, Z -6.3333, A 0.000, B 0.000, C 0.000 }
gfCNCPoint5[4566] = {X 517.3058, Y 36.7738, Z -6.3333, A 0.000, B 0.000, C 0.000 }
gfCNCPoint5[4567] = {X 518.0643, Y 36.2972, Z -6.3333, A 0.000, B 0.000, C 0.000 }
gfCNCPoint5[4568] = {X 518.9097, Y 36.0014, Z -6.3333, A 0.000, B 0.000, C 0.000 }
gfCNCPoint5[4569] = {X 519.7998, Y 35.9011, Z -6.3333, A 0.000, B 0.000, C 0.000 }
gfCNCPoint5[4570] = {X 520.5225, Y 35.9015, Z -6.3333, A 0.000, B 0.000, C 0.000 }
gfCNCPoint5[4571] = {X 521.3205, Y 35.9930, Z -6.3333, A 0.000, B 0.000, C 0.000 }
gfCNCPoint5[4572] = {X 522.0840, Y 36.2420, Z -6.3333, A 0.000, B 0.000, C 0.000 }
gfCNCPoint5[4573] = {X 522.7825, Y 36.6386, Z -6.3333, A 0.000, B 0.000, C 0.000 }
gfCNCPoint5[4574] = {X 523.3876, Y 37.1667, Z -6.3333, A 0.000, B 0.000, C 0.000 }
gfCNCPoint5[4575] = {X 523.8750, Y 37.8050, Z -6.3333, A 0.000, B 0.000, C 0.000 }
gfCNCPoint5[4576] = {X 534.9519, Y 37.8054, Z -6.3333, A 0.000, B 0.000, C 0.000 }
gfCNCPoint5[4577] = {X 534.9519, Y 33.6460, Z -6.3333, A 0.000, B 0.000, C 0.000 }
gfCNCPoint5[4578] = {X 529.9337, Y 33.6457, Z -6.3333, A 0.000, B 0.000, C 0.000 }
gfCNCPoint5[4579] = {X 529.8224, Y 33.8188, Z -6.3333, A 0.000, B 0.000, C 0.000 }
gfCNCPoint5[4580] = {X 529.1829, Y 34.5417, Z -6.3333, A 0.000, B 0.000, C 0.000 }
gfCNCPoint5[4581] = {X 528.3889, Y 35.0905, Z -6.3333, A 0.000, B 0.000, C 0.000 }
gfCNCPoint5[4582] = {X 527.4865, Y 35.4330, Z -6.3333, A 0.000, B 0.000, C 0.000 }
gfCNCPoint5[4583] = {X 526.5283, Y 35.5495, Z -6.3333, A 0.000, B 0.000, C 0.000 }
gfCNCPoint5[4584] = {X 525.8868, Y 35.5495, Z -6.3333, A 0.000, B 0.000, C 0.000 }
gfCNCPoint5[4585] = {X 524.9967, Y 35.4492, Z -6.3333, A 0.000, B 0.000, C 0.000 }
gfCNCPoint5[4586] = {X 524.1512, Y 35.1533, Z -6.3333, A 0.000, B 0.000, C 0.000 }
gfCNCPoint5[4587] = {X 523.3928, Y 34.6768, Z -6.3333, A 0.000, B 0.000, C 0.000 }
gfCNCPoint5[4588] = {X 522.7594, Y 34.0434, Z -6.3333, A 0.000, B 0.000, C 0.000 }
gfCNCPoint5[4589] = {X 522.2829, Y 33.2850, Z -6.3333, A 0.000, B 0.000, C 0.000 }
gfCNCPoint5[4590] = {X 521.9870, Y 32.4395, Z -6.3333, A 0.000, B 0.000, C 0.000 }
gfCNCPoint5[4591] = {X 521.8868, Y 31.5495, Z -6.3333, A 0.000, B 0.000, C 0.000 }
gfCNCPoint5[4592] = {X 521.8868, Y 24.5714, Z -6.3333, A 0.000, B 0.000, C 0.000 }
gfCNCPoint5[4593] = {X 521.9870, Y 23.6813, Z -6.3333, A 0.000, B 0.000, C 0.000 }
gfCNCPoint5[4594] = {X 522.2829, Y 22.8359, Z -6.3333, A 0.000, B 0.000, C 0.000 }
gfCNCPoint5[4595] = {X 522.7594, Y 22.0775, Z -6.3333, A 0.000, B 0.000, C 0.000 }
gfCNCPoint5[4596] = {X 523.3928, Y 21.4441, Z -6.3333, A 0.000, B 0.000, C 0.000 }
gfCNCPoint5[4597] = {X 524.1512, Y 20.9675, Z -6.3333, A 0.000, B 0.000, C 0.000 }
gfCNCPoint5[4598] = {X 524.9967, Y 20.6717, Z -6.3333, A 0.000, B 0.000, C 0.000 }
gfCNCPoint5[4599] = {X 525.8868, Y 20.5714, Z -6.3333, A 0.000, B 0.000, C 0.000 }
gfCNCPoint5[4600] = {X 526.5664, Y 20.5716, Z -6.3333, A 0.000, B 0.000, C 0.000 }
gfCNCPoint5[4601] = {X 527.3628, Y 20.6594, Z -6.3333, A 0.000, B 0.000, C 0.000 }
gfCNCPoint5[4602] = {X 528.1258, Y 20.9042, Z -6.3333, A 0.000, B 0.000, C 0.000 }
gfCNCPoint5[4603] = {X 528.8246, Y 21.2961, Z -6.3333, A 0.000, B 0.000, C 0.000 }
gfCNCPoint5[4604] = {X 529.4313, Y 21.8195, Z -6.3333, A 0.000, B 0.000, C 0.000 }
gfCNCPoint5[4605] = {X 529.9215, Y 22.4532, Z -6.3333, A 0.000, B 0.000, C 0.000 }
gfCNCPoint5[4606] = {X 534.9519, Y 22.4534, Z -6.3333, A 0.000, B 0.000, C 0.000 }
gfCNCPoint5[4607] = {X 534.9519, Y 19.7824, Z -6.3333, A 0.000, B 0.000, C 0.000 }
gfCNCPoint5[4608] = {X 534.9520, Y 19.3824, Z -6.3333, A 0.000, B 0.000, C 0.000 }
gfCNCPoint5[4609] = {X 524.0171, Y 19.3822, Z -6.3333, A 0.000, B 0.000, C 0.000 }
gfCNCPoint5[4610] = {X 523.9046, Y 19.5552, Z -6.3333, A 0.000, B 0.000, C 0.000 }
gfCNCPoint5[4611] = {X 523.2651, Y 20.2781, Z -6.3333, A 0.000, B 0.000, C 0.000 }
gfCNCPoint5[4612] = {X 522.4711, Y 20.8268, Z -6.3333, A 0.000, B 0.000, C 0.000 }
gfCNCPoint5[4613] = {X 521.5688, Y 21.1693, Z -6.3333, A 0.000, B 0.000, C 0.000 }
gfCNCPoint5[4614] = {X 520.6107, Y 21.2857, Z -6.3333, A 0.000, B 0.000, C 0.000 }
gfCNCPoint5[4615] = {X 519.9691, Y 21.2857, Z -6.3333, A 0.000, B 0.000, C 0.000 }
gfCNCPoint5[4616] = {X 519.0790, Y 21.1854, Z -6.3333, A 0.000, B 0.000, C 0.000 }
gfCNCPoint5[4617] = {X 518.2336, Y 20.8896, Z -6.3333, A 0.000, B 0.000, C 0.000 }
gfCNCPoint5[4618] = {X 517.4751, Y 20.4130, Z -6.3333, A 0.000, B 0.000, C 0.000 }
gfCNCPoint5[4619] = {X 516.8418, Y 19.7797, Z -6.3333, A 0.000, B 0.000, C 0.000 }
gfCNCPoint5[4620] = {X 516.3652, Y 19.0212, Z -6.3333, A 0.000, B 0.000, C 0.000 }
gfCNCPoint5[4621] = {X 516.0694, Y 18.1758, Z -6.3333, A 0.000, B 0.000, C 0.000 }
gfCNCPoint5[4622] = {X 515.9691, Y 17.2857, Z -6.3333, A 0.000, B 0.000, C 0.000 }
gfCNCPoint5[4623] = {X 515.9691, Y 10.3077, Z -6.3333, A 0.000, B 0.000, C 0.000 }
gfCNCPoint5[4624] = {X 516.0694, Y 9.4176, Z -6.3333, A 0.000, B 0.000, C 0.000 }
gfCNCPoint5[4625] = {X 516.3652, Y 8.5721, Z -6.3333, A 0.000, B 0.000, C 0.000 }
gfCNCPoint5[4626] = {X 516.8418, Y 7.8137, Z -6.3333, A 0.000, B 0.000, C 0.000 }
gfCNCPoint5[4627] = {X 517.4752, Y 7.1803, Z -6.3333, A 0.000, B 0.000, C 0.000 }
gfCNCPoint5[4628] = {X 518.2336, Y 6.7038, Z -6.3333, A 0.000, B 0.000, C 0.000 }
gfCNCPoint5[4629] = {X 519.0791, Y 6.4080, Z -6.3333, A 0.000, B 0.000, C 0.000 }
gfCNCPoint5[4630] = {X 519.9692, Y 6.3077, Z -6.3333, A 0.000, B 0.000, C 0.000 }
gfCNCPoint5[4631] = {X 520.6472, Y 6.3079, Z -6.3333, A 0.000, B 0.000, C 0.000 }
gfCNCPoint5[4632] = {X 521.4440, Y 6.3954, Z -6.3333, A 0.000, B 0.000, C 0.000 }
gfCNCPoint5[4633] = {X 522.2073, Y 6.6401, Z -6.3333, A 0.000, B 0.000, C 0.000 }
gfCNCPoint5[4634] = {X 522.9065, Y 7.0321, Z -6.3333, A 0.000, B 0.000, C 0.000 }
gfCNCPoint5[4635] = {X 523.5135, Y 7.5555, Z -6.3333, A 0.000, B 0.000, C 0.000 }
gfCNCPoint5[4636] = {X 524.0039, Y 8.1895, Z -6.3333, A 0.000, B 0.000, C 0.000 }
gfCNCPoint5[4637] = {X 533.9634, Y 8.1897, Z -6.3333, A 0.000, B 0.000, C 0.000 }
gfCNCPoint5[4638] = {X 533.9635, Y 4.1097, Z -6.3333, A 0.000, B 0.000, C 0.000 }
gfCNCPoint5[4639] = {X 533.9635, Y 4.1097, Z -3.3333, A 0.000, B 0.000, C 0.000 }
gfCNCPoint5[4640] = {X 533.9635, Y 4.1097, Z 11.0000, A 0.000, B 0.000, C 0.000 }
gfCNCPoint5[4641] = {X 419.6147, Y 26.5282, Z 11.0000, A 0.000, B 0.000, C 0.000 }
gfCNCPoint5[4642] = {X 419.6147, Y 26.5282, Z -3.3333, A 0.000, B 0.000, C 0.000 }
gfCNCPoint5[4643] = {X 419.6147, Y 26.5282, Z -6.3333, A 0.000, B 0.000, C 0.000 }
gfCNCPoint5[4644] = {X 416.1512, Y 24.3717, Z -6.3333, A 0.000, B 0.000, C 0.000 }
gfCNCPoint5[4645] = {X 411.5476, Y 31.7653, Z -6.3333, A 0.000, B 0.000, C 0.000 }
gfCNCPoint5[4646] = {X 411.5482, Y 40.8977, Z -6.3333, A 0.000, B 0.000, C 0.000 }
gfCNCPoint5[4647] = {X 412.1864, Y 41.5836, Z -6.3333, A 0.000, B 0.000, C 0.000 }
gfCNCPoint5[4648] = {X 412.6665, Y 42.3881, Z -6.3333, A 0.000, B 0.000, C 0.000 }
gfCNCPoint5[4649] = {X 412.9670, Y 43.2755, Z -6.3333, A 0.000, B 0.000, C 0.000 }
gfCNCPoint5[4650] = {X 413.0747, Y 44.2062, Z -6.3333, A 0.000, B 0.000, C 0.000 }
gfCNCPoint5[4651] = {X 413.0747, Y 45.0002, Z -6.3333, A 0.000, B 0.000, C 0.000 }
gfCNCPoint5[4652] = {X 412.9663, Y 45.9614, Z -6.3333, A 0.000, B 0.000, C 0.000 }
gfCNCPoint5[4653] = {X 412.6468, Y 46.8745, Z -6.3333, A 0.000, B 0.000, C 0.000 }
gfCNCPoint5[4654] = {X 412.1321, Y 47.6936, Z -6.3333, A 0.000, B 0.000, C 0.000 }
gfCNCPoint5[4655] = {X 411.4481, Y 48.3776, Z -6.3333, A 0.000, B 0.000, C 0.000 }
gfCNCPoint5[4656] = {X 410.6290, Y 48.8922, Z -6.3333, A 0.000, B 0.000, C 0.000 }
gfCNCPoint5[4657] = {X 409.7159, Y 49.2117, Z -6.3333, A 0.000, B 0.000, C 0.000 }
gfCNCPoint5[4658] = {X 408.7547, Y 49.3200, Z -6.3333, A 0.000, B 0.000, C 0.000 }
gfCNCPoint5[4659] = {X 402.3112, Y 49.3200, Z -6.3333, A 0.000, B 0.000, C 0.000 }
gfCNCPoint5[4660] = {X 401.3546, Y 49.2127, Z -6.3333, A 0.000, B 0.000, C 0.000 }
gfCNCPoint5[4661] = {X 400.4455, Y 48.8963, Z -6.3333, A 0.000, B 0.000, C 0.000 }
gfCNCPoint5[4662] = {X 399.6290, Y 48.3864, Z -6.3333, A 0.000, B 0.000, C 0.000 }
gfCNCPoint5[4663] = {X 398.9457, Y 47.7084, Z -6.3333, A 0.000, B 0.000, C 0.000 }
gfCNCPoint5[4664] = {X 398.4295, Y 46.8959, Z -6.3333, A 0.000, B 0.000, C 0.000 }
gfCNCPoint5[4665] = {X 398.1060, Y 45.9892, Z -6.3333, A 0.000, B 0.000, C 0.000 }
gfCNCPoint5[4666] = {X 397.9913, Y 45.0335, Z -6.3333, A 0.000, B 0.000, C 0.000 }
gfCNCPoint5[4667] = {X 397.9916, Y 44.1528, Z -6.3333, A 0.000, B 0.000, C 0.000 }
gfCNCPoint5[4668] = {X 398.1015, Y 43.2391, Z -6.3333, A 0.000, B 0.000, C 0.000 }
gfCNCPoint5[4669] = {X 398.4024, Y 42.3694, Z -6.3333, A 0.000, B 0.000, C 0.000 }
gfCNCPoint5[4670] = {X 398.8807, Y 41.5832, Z -6.3333, A 0.000, B 0.000, C 0.000 }
gfCNCPoint5[4671] = {X 399.5147, Y 40.9161, Z -6.3333, A 0.000, B 0.000, C 0.000 }
gfCNCPoint5[4672] = {X 399.4729, Y 31.6017, Z -6.3333, A 0.000, B 0.000, C 0.000 }
gfCNCPoint5[4673] = {X 393.5202, Y 21.2501, Z -6.3333, A 0.000, B 0.000, C 0.000 }
gfCNCPoint5[4674] = {X 392.6316, Y 19.7382, Z -6.3333, A 0.000, B 0.000, C 0.000 }
gfCNCPoint5[4675] = {X 391.7143, Y 18.2434, Z -6.3333, A 0.000, B 0.000, C 0.000 }
gfCNCPoint5[4676] = {X 391.2311, Y 17.5711, Z -6.3333, A 0.000, B 0.000, C 0.000 }
gfCNCPoint5[4677] = {X 390.6668, Y 16.9652, Z -6.3333, A 0.000, B 0.000, C 0.000 }
gfCNCPoint5[4678] = {X 389.7901, Y 16.4728, Z -6.3333, A 0.000, B 0.000, C 0.000 }
gfCNCPoint5[4679] = {X 389.0510, Y 15.7910, Z -6.3333, A 0.000, B 0.000, C 0.000 }
gfCNCPoint5[4680] = {X 388.4895, Y 14.9569, Z -6.3333, A 0.000, B 0.000, C 0.000 }
gfCNCPoint5[4681] = {X 388.1361, Y 14.0156, Z -6.3333, A 0.000, B 0.000, C 0.000 }
gfCNCPoint5[4682] = {X 388.0098, Y 13.0180, Z -6.3333, A 0.000, B 0.000, C 0.000 }
gfCNCPoint5[4683] = {X 388.0096, Y 12.1868, Z -6.3333, A 0.000, B 0.000, C 0.000 }
gfCNCPoint5[4684] = {X 388.1179, Y 11.2255, Z -6.3333, A 0.000, B 0.000, C 0.000 }
gfCNCPoint5[4685] = {X 388.4374, Y 10.3125, Z -6.3333, A 0.000, B 0.000, C 0.000 }
gfCNCPoint5[4686] = {X 388.9521, Y 9.4933, Z -6.3333, A 0.000, B 0.000, C 0.000 }
gfCNCPoint5[4687] = {X 389.6361, Y 8.8093, Z -6.3333, A 0.000, B 0.000, C 0.000 }
gfCNCPoint5[4688] = {X 390.4552, Y 8.2946, Z -6.3333, A 0.000, B 0.000, C 0.000 }
gfCNCPoint5[4689] = {X 391.3683, Y 7.9751, Z -6.3333, A 0.000, B 0.000, C 0.000 }
gfCNCPoint5[4690] = {X 392.3296, Y 7.8668, Z -6.3333, A 0.000, B 0.000, C 0.000 }
gfCNCPoint5[4691] = {X 399.1118, Y 7.8668, Z -6.3333, A 0.000, B 0.000, C 0.000 }
gfCNCPoint5[4692] = {X 400.0730, Y 7.9751, Z -6.3333, A 0.000, B 0.000, C 0.000 }
gfCNCPoint5[4693] = {X 400.9861, Y 8.2946, Z -6.3333, A 0.000, B 0.000, C 0.000 }
gfCNCPoint5[4694] = {X 401.8052, Y 8.8093, Z -6.3333, A 0.000, B 0.000, C 0.000 }
gfCNCPoint5[4695] = {X 402.4893, Y 9.4933, Z -6.3333, A 0.000, B 0.000, C 0.000 }
gfCNCPoint5[4696] = {X 403.0039, Y 10.3124, Z -6.3333, A 0.000, B 0.000, C 0.000 }
gfCNCPoint5[4697] = {X 403.3234, Y 11.2255, Z -6.3333, A 0.000, B 0.000, C 0.000 }
gfCNCPoint5[4698] = {X 403.4318, Y 12.1868, Z -6.3333, A 0.000, B 0.000, C 0.000 }
gfCNCPoint5[4699] = {X 403.4318, Y 12.9782, Z -6.3333, A 0.000, B 0.000, C 0.000 }
gfCNCPoint5[4700] = {X 403.3293, Y 13.9134, Z -6.3333, A 0.000, B 0.000, C 0.000 }
gfCNCPoint5[4701] = {X 403.0267, Y 14.8044, Z -6.3333, A 0.000, B 0.000, C 0.000 }
gfCNCPoint5[4702] = {X 405.3559, Y 18.8226, Z -6.3333, A 0.000, B 0.000, C 0.000 }
gfCNCPoint5[4703] = {X 407.8732, Y 14.7534, Z -6.3333, A 0.000, B 0.000, C 0.000 }
gfCNCPoint5[4704] = {X 407.5920, Y 13.9041, Z -6.3333, A 0.000, B 0.000, C 0.000 }
gfCNCPoint5[4705] = {X 407.4917, Y 13.0151, Z -6.3333, A 0.000, B 0.000, C 0.000 }
gfCNCPoint5[4706] = {X 407.4915, Y 12.1868, Z -6.3333, A 0.000, B 0.000, C 0.000 }
gfCNCPoint5[4707] = {X 407.5999, Y 11.2255, Z -6.3333, A 0.000, B 0.000, C 0.000 }
gfCNCPoint5[4708] = {X 407.9194, Y 10.3124, Z -6.3333, A 0.000, B 0.000, C 0.000 }
gfCNCPoint5[4709] = {X 408.4340, Y 9.4933, Z -6.3333, A 0.000, B 0.000, C 0.000 }
gfCNCPoint5[4710] = {X 409.1181, Y 8.8093, Z -6.3333, A 0.000, B 0.000, C 0.000 }
gfCNCPoint5[4711] = {X 409.9372, Y 8.2946, Z -6.3333, A 0.000, B 0.000, C 0.000 }
gfCNCPoint5[4712] = {X 410.8502, Y 7.9751, Z -6.3333, A 0.000, B 0.000, C 0.000 }
gfCNCPoint5[4713] = {X 411.8115, Y 7.8668, Z -6.3333, A 0.000, B 0.000, C 0.000 }
gfCNCPoint5[4714] = {X 419.3245, Y 7.8668, Z -6.3333, A 0.000, B 0.000, C 0.000 }
gfCNCPoint5[4715] = {X 420.2858, Y 7.9751, Z -6.3333, A 0.000, B 0.000, C 0.000 }
gfCNCPoint5[4716] = {X 421.1988, Y 8.2946, Z -6.3333, A 0.000, B 0.000, C 0.000 }
gfCNCPoint5[4717] = {X 422.0179, Y 8.8093, Z -6.3333, A 0.000, B 0.000, C 0.000 }
gfCNCPoint5[4718] = {X 422.7020, Y 9.4933, Z -6.3333, A 0.000, B 0.000, C 0.000 }
gfCNCPoint5[4719] = {X 423.2166, Y 10.3124, Z -6.3333, A 0.000, B 0.000, C 0.000 }
gfCNCPoint5[4720] = {X 423.5361, Y 11.2255, Z -6.3333, A 0.000, B 0.000, C 0.000 }
gfCNCPoint5[4721] = {X 423.6445, Y 12.1868, Z -6.3333, A 0.000, B 0.000, C 0.000 }
gfCNCPoint5[4722] = {X 423.6445, Y 12.9802, Z -6.3333, A 0.000, B 0.000, C 0.000 }
gfCNCPoint5[4723] = {X 423.5518, Y 13.8468, Z -6.3333, A 0.000, B 0.000, C 0.000 }
gfCNCPoint5[4724] = {X 423.2895, Y 14.6779, Z -6.3333, A 0.000, B 0.000, C 0.000 }
gfCNCPoint5[4725] = {X 422.8680, Y 15.4406, Z -6.3333, A 0.000, B 0.000, C 0.000 }
gfCNCPoint5[4726] = {X 422.3037, Y 16.1049, Z -6.3333, A 0.000, B 0.000, C 0.000 }
gfCNCPoint5[4727] = {X 421.6192, Y 16.6443, Z -6.3333, A 0.000, B 0.000, C 0.000 }
gfCNCPoint5[4728] = {X 420.8415, Y 17.0376, Z -6.3333, A 0.000, B 0.000, C 0.000 }
gfCNCPoint5[4729] = {X 420.1251, Y 18.0009, Z -6.3333, A 0.000, B 0.000, C 0.000 }
gfCNCPoint5[4730] = {X 419.4769, Y 19.0115, Z -6.3333, A 0.000, B 0.000, C 0.000 }
gfCNCPoint5[4731] = {X 417.9942, Y 21.4117, Z -6.3333, A 0.000, B 0.000, C 0.000 }
gfCNCPoint5[4732] = {X 416.1512, Y 24.3717, Z -6.3333, A 0.000, B 0.000, C 0.000 }
gfCNCPoint5[4733] = {X 419.5468, Y 26.4859, Z -6.3333, A 0.000, B 0.000, C 0.000 }
gfCNCPoint5[4734] = {X 416.0833, Y 24.3294, Z -6.3333, A 0.000, B 0.000, C 0.000 }
gfCNCPoint5[4735] = {X 411.4676, Y 31.7424, Z -6.3333, A 0.000, B 0.000, C 0.000 }
gfCNCPoint5[4736] = {X 411.4682, Y 40.9343, Z -6.3333, A 0.000, B 0.000, C 0.000 }
gfCNCPoint5[4737] = {X 412.1060, Y 41.6099, Z -6.3333, A 0.000, B 0.000, C 0.000 }
gfCNCPoint5[4738] = {X 412.5862, Y 42.4052, Z -6.3333, A 0.000, B 0.000, C 0.000 }
gfCNCPoint5[4739] = {X 412.8870, Y 43.2842, Z -6.3333, A 0.000, B 0.000, C 0.000 }
gfCNCPoint5[4740] = {X 412.9947, Y 44.2070, Z -6.3333, A 0.000, B 0.000, C 0.000 }
gfCNCPoint5[4741] = {X 412.9947, Y 45.0002, Z -6.3333, A 0.000, B 0.000, C 0.000 }
gfCNCPoint5[4742] = {X 412.8883, Y 45.9436, Z -6.3333, A 0.000, B 0.000, C 0.000 }
gfCNCPoint5[4743] = {X 412.5747, Y 46.8398, Z -6.3333, A 0.000, B 0.000, C 0.000 }
gfCNCPoint5[4744] = {X 412.0696, Y 47.6437, Z -6.3333, A 0.000, B 0.000, C 0.000 }
gfCNCPoint5[4745] = {X 411.3982, Y 48.3150, Z -6.3333, A 0.000, B 0.000, C 0.000 }
gfCNCPoint5[4746] = {X 410.5943, Y 48.8201, Z -6.3333, A 0.000, B 0.000, C 0.000 }
gfCNCPoint5[4747] = {X 409.6981, Y 49.1337, Z -6.3333, A 0.000, B 0.000, C 0.000 }
gfCNCPoint5[4748] = {X 408.7547, Y 49.2400, Z -6.3333, A 0.000, B 0.000, C 0.000 }
gfCNCPoint5[4749] = {X 402.3112, Y 49.2400, Z -6.3333, A 0.000, B 0.000, C 0.000 }
gfCNCPoint5[4750] = {X 401.3723, Y 49.1347, Z -6.3333, A 0.000, B 0.000, C 0.000 }
gfCNCPoint5[4751] = {X 400.4800, Y 48.8242, Z -6.3333, A 0.000, B 0.000, C 0.000 }
gfCNCPoint5[4752] = {X 399.6786, Y 48.3237, Z -6.3333, A 0.000, B 0.000, C 0.000 }
gfCNCPoint5[4753] = {X 399.0080, Y 47.6582, Z -6.3333, A 0.000, B 0.000, C 0.000 }
gfCNCPoint5[4754] = {X 398.5013, Y 46.8608, Z -6.3333, A 0.000, B 0.000, C 0.000 }
gfCNCPoint5[4755] = {X 398.1839, Y 45.9709, Z -6.3333, A 0.000, B 0.000, C 0.000 }
gfCNCPoint5[4756] = {X 398.0713, Y 45.0329, Z -6.3333, A 0.000, B 0.000, C 0.000 }
gfCNCPoint5[4757] = {X 398.0716, Y 44.1538, Z -6.3333, A 0.000, B 0.000, C 0.000 }
gfCNCPoint5[4758] = {X 398.1815, Y 43.2480, Z -6.3333, A 0.000, B 0.000, C 0.000 }
gfCNCPoint5[4759] = {X 398.4827, Y 42.3867, Z -6.3333, A 0.000, B 0.000, C 0.000 }
gfCNCPoint5[4760] = {X 398.9612, Y 41.6098, Z -6.3333, A 0.000, B 0.000, C 0.000 }
gfCNCPoint5[4761] = {X 399.5948, Y 40.9532, Z -6.3333, A 0.000, B 0.000, C 0.000 }
gfCNCPoint5[4762] = {X 399.5528, Y 31.5801, Z -6.3333, A 0.000, B 0.000, C 0.000 }
gfCNCPoint5[4763] = {X 393.5896, Y 21.2102, Z -6.3333, A 0.000, B 0.000, C 0.000 }
gfCNCPoint5[4764] = {X 392.7001, Y 19.6970, Z -6.3333, A 0.000, B 0.000, C 0.000 }
gfCNCPoint5[4765] = {X 391.7821, Y 18.2009, Z -6.3333, A 0.000, B 0.000, C 0.000 }
gfCNCPoint5[4766] = {X 391.2883, Y 17.5146, Z -6.3333, A 0.000, B 0.000, C 0.000 }
gfCNCPoint5[4767] = {X 390.7110, Y 16.8969, Z -6.3333, A 0.000, B 0.000, C 0.000 }
gfCNCPoint5[4768] = {X 389.8466, Y 16.4149, Z -6.3333, A 0.000, B 0.000, C 0.000 }
gfCNCPoint5[4769] = {X 389.1174, Y 15.7456, Z -6.3333, A 0.000, B 0.000, C 0.000 }
gfCNCPoint5[4770] = {X 388.5633, Y 14.9254, Z -6.3333, A 0.000, B 0.000, C 0.000 }
gfCNCPoint5[4771] = {X 388.2144, Y 13.9992, Z -6.3333, A 0.000, B 0.000, C 0.000 }
gfCNCPoint5[4772] = {X 388.0898, Y 13.0173, Z -6.3333, A 0.000, B 0.000, C 0.000 }
gfCNCPoint5[4773] = {X 388.0896, Y 12.1868, Z -6.3333, A 0.000, B 0.000, C 0.000 }
gfCNCPoint5[4774] = {X 388.1959, Y 11.2433, Z -6.3333, A 0.000, B 0.000, C 0.000 }
gfCNCPoint5[4775] = {X 388.5095, Y 10.3472, Z -6.3333, A 0.000, B 0.000, C 0.000 }
gfCNCPoint5[4776] = {X 389.0147, Y 9.5432, Z -6.3333, A 0.000, B 0.000, C 0.000 }
gfCNCPoint5[4777] = {X 389.6860, Y 8.8719, Z -6.3333, A 0.000, B 0.000, C 0.000 }
gfCNCPoint5[4778] = {X 390.4900, Y 8.3667, Z -6.3333, A 0.000, B 0.000, C 0.000 }
gfCNCPoint5[4779] = {X 391.3861, Y 8.0531, Z -6.3333, A 0.000, B 0.000, C 0.000 }
gfCNCPoint5[4780] = {X 392.3296, Y 7.9468, Z -6.3333, A 0.000, B 0.000, C 0.000 }
gfCNCPoint5[4781] = {X 399.1118, Y 7.9468, Z -6.3333, A 0.000, B 0.000, C 0.000 }
gfCNCPoint5[4782] = {X 400.0552, Y 8.0531, Z -6.3333, A 0.000, B 0.000, C 0.000 }
gfCNCPoint5[4783] = {X 400.9514, Y 8.3667, Z -6.3333, A 0.000, B 0.000, C 0.000 }
gfCNCPoint5[4784] = {X 401.7554, Y 8.8718, Z -6.3333, A 0.000, B 0.000, C 0.000 }
gfCNCPoint5[4785] = {X 402.4267, Y 9.5432, Z -6.3333, A 0.000, B 0.000, C 0.000 }
gfCNCPoint5[4786] = {X 402.9319, Y 10.3471, Z -6.3333, A 0.000, B 0.000, C 0.000 }
gfCNCPoint5[4787] = {X 403.2455, Y 11.2433, Z -6.3333, A 0.000, B 0.000, C 0.000 }
gfCNCPoint5[4788] = {X 403.3518, Y 12.1868, Z -6.3333, A 0.000, B 0.000, C 0.000 }
gfCNCPoint5[4789] = {X 403.3518, Y 12.9782, Z -6.3333, A 0.000, B 0.000, C 0.000 }
gfCNCPoint5[4790] = {X 403.2466, Y 13.9164, Z -6.3333, A 0.000, B 0.000, C 0.000 }
gfCNCPoint5[4791] = {X 402.9364, Y 14.8081, Z -6.3333, A 0.000, B 0.000, C 0.000 }
gfCNCPoint5[4792] = {X 405.3536, Y 18.9783, Z -6.3333, A 0.000, B 0.000, C 0.000 }
gfCNCPoint5[4793] = {X 407.9638, Y 14.7591, Z -6.3333, A 0.000, B 0.000, C 0.000 }
gfCNCPoint5[4794] = {X 407.6747, Y 13.9077, Z -6.3333, A 0.000, B 0.000, C 0.000 }
gfCNCPoint5[4795] = {X 407.5717, Y 13.0144, Z -6.3333, A 0.000, B 0.000, C 0.000 }
gfCNCPoint5[4796] = {X 407.5715, Y 12.1868, Z -6.3333, A 0.000, B 0.000, C 0.000 }
gfCNCPoint5[4797] = {X 407.6778, Y 11.2433, Z -6.3333, A 0.000, B 0.000, C 0.000 }
gfCNCPoint5[4798] = {X 407.9914, Y 10.3471, Z -6.3333, A 0.000, B 0.000, C 0.000 }
gfCNCPoint5[4799] = {X 408.4966, Y 9.5432, Z -6.3333, A 0.000, B 0.000, C 0.000 }
gfCNCPoint5[4800] = {X 409.1679, Y 8.8718, Z -6.3333, A 0.000, B 0.000, C 0.000 }
gfCNCPoint5[4801] = {X 409.9719, Y 8.3667, Z -6.3333, A 0.000, B 0.000, C 0.000 }
gfCNCPoint5[4802] = {X 410.8680, Y 8.0531, Z -6.3333, A 0.000, B 0.000, C 0.000 }
gfCNCPoint5[4803] = {X 411.8115, Y 7.9468, Z -6.3333, A 0.000, B 0.000, C 0.000 }
gfCNCPoint5[4804] = {X 419.3245, Y 7.9468, Z -6.3333, A 0.000, B 0.000, C 0.000 }
gfCNCPoint5[4805] = {X 420.2679, Y 8.0531, Z -6.3333, A 0.000, B 0.000, C 0.000 }
gfCNCPoint5[4806] = {X 421.1641, Y 8.3667, Z -6.3333, A 0.000, B 0.000, C 0.000 }
gfCNCPoint5[4807] = {X 421.9681, Y 8.8718, Z -6.3333, A 0.000, B 0.000, C 0.000 }
gfCNCPoint5[4808] = {X 422.6394, Y 9.5432, Z -6.3333, A 0.000, B 0.000, C 0.000 }
gfCNCPoint5[4809] = {X 423.1446, Y 10.3471, Z -6.3333, A 0.000, B 0.000, C 0.000 }
gfCNCPoint5[4810] = {X 423.4582, Y 11.2433, Z -6.3333, A 0.000, B 0.000, C 0.000 }
gfCNCPoint5[4811] = {X 423.5645, Y 12.1868, Z -6.3333, A 0.000, B 0.000, C 0.000 }
gfCNCPoint5[4812] = {X 423.5645, Y 12.9796, Z -6.3333, A 0.000, B 0.000, C 0.000 }
gfCNCPoint5[4813] = {X 423.4728, Y 13.8339, Z -6.3333, A 0.000, B 0.000, C 0.000 }
gfCNCPoint5[4814] = {X 423.2132, Y 14.6529, Z -6.3333, A 0.000, B 0.000, C 0.000 }
gfCNCPoint5[4815] = {X 422.7960, Y 15.4040, Z -6.3333, A 0.000, B 0.000, C 0.000 }
gfCNCPoint5[4816] = {X 422.2379, Y 16.0572, Z -6.3333, A 0.000, B 0.000, C 0.000 }
gfCNCPoint5[4817] = {X 421.5611, Y 16.5865, Z -6.3333, A 0.000, B 0.000, C 0.000 }
gfCNCPoint5[4818] = {X 420.7926, Y 16.9707, Z -6.3333, A 0.000, B 0.000, C 0.000 }
gfCNCPoint5[4819] = {X 420.0657, Y 17.9462, Z -6.3333, A 0.000, B 0.000, C 0.000 }
gfCNCPoint5[4820] = {X 419.4085, Y 18.9700, Z -6.3333, A 0.000, B 0.000, C 0.000 }
gfCNCPoint5[4821] = {X 417.9262, Y 21.3695, Z -6.3333, A 0.000, B 0.000, C 0.000 }
gfCNCPoint5[4822] = {X 416.0833, Y 24.3294, Z -6.3333, A 0.000, B 0.000, C 0.000 }
gfCNCPoint5[4823] = {X 419.4789, Y 26.4436, Z -6.3333, A 0.000, B 0.000, C 0.000 }
gfCNCPoint5[4824] = {X 416.0154, Y 24.2871, Z -6.3333, A 0.000, B 0.000, C 0.000 }
gfCNCPoint5[4825] = {X 411.3876, Y 31.7196, Z -6.3333, A 0.000, B 0.000, C 0.000 }
gfCNCPoint5[4826] = {X 411.3882, Y 40.9714, Z -6.3333, A 0.000, B 0.000, C 0.000 }
gfCNCPoint5[4827] = {X 412.0256, Y 41.6364, Z -6.3333, A 0.000, B 0.000, C 0.000 }
gfCNCPoint5[4828] = {X 412.5059, Y 42.4224, Z -6.3333, A 0.000, B 0.000, C 0.000 }
gfCNCPoint5[4829] = {X 412.8069, Y 43.2929, Z -6.3333, A 0.000, B 0.000, C 0.000 }
gfCNCPoint5[4830] = {X 412.9147, Y 44.2077, Z -6.3333, A 0.000, B 0.000, C 0.000 }
gfCNCPoint5[4831] = {X 412.9147, Y 45.0002, Z -6.3333, A 0.000, B 0.000, C 0.000 }
gfCNCPoint5[4832] = {X 412.8103, Y 45.9258, Z -6.3333, A 0.000, B 0.000, C 0.000 }
gfCNCPoint5[4833] = {X 412.5027, Y 46.8051, Z -6.3333, A 0.000, B 0.000, C 0.000 }
gfCNCPoint5[4834] = {X 412.0070, Y 47.5938, Z -6.3333, A 0.000, B 0.000, C 0.000 }
